// TwinCAT 3 PLC project rixs_optics_sim
// ProgramVersion: 3.1.4022.7
// libraries:
//   lcls2-cc-lib, * (SLAC)
//   PMPS, * (SLAC - LCLS)
//   Tc2_MC2, * (Beckhoff Automation GmbH)
//   Tc2_SerialCom, * (Beckhoff Automation GmbH)
//   Tc2_Standard, * (Beckhoff Automation GmbH)
//   Tc2_System, * (Beckhoff Automation GmbH)
//   Tc2_TcpIp, * (Beckhoff Automation GmbH)
//   Tc2_Utilities, * (Beckhoff Automation GmbH)
//   Tc3_Module, * (Beckhoff Automation GmbH)
//   LCLS General,newest,SLAC
//   lcls-twincat-motion,newest,SLAC
//   lcls-twincat-optics,newest,SLAC
// project tree:
//   DUTs/ ENUM_XS_YAG_States.TcDUT (not stored)
//   Function Blocks/ FB_XS_YAG_States.TcPOU (not stored)
//   GVLs/ GVL_COM_Buffers.TcGVL (not stored), GVL_M1K1.TcGVL (not stored), GVL_M1K1_BENDER_Constants.TcGVL (not stored), GVL_M1K1_BENDER_RTD.TcGVL (not stored), GVL_M1K1_Constants.TcGVL (not stored), GVL_M1K2.TcGVL (not stored), GVL_M1K2_Constants.TcGVL (not stored), GVL_PMPS.TcGVL, GVL_SerialIO.TcGVL (not stored), Main.TcGVL
//   / PiezoDriver.TcTTO (not stored), PlcTask.TcTTO (not stored), SerialIO.TcTTO (not stored)
//   POUs/DAQ Comm/ DUT_01_Channel_NW.TcDUT (not stored), DUT_Channel_NW.TcDUT (not stored), DUT_Header_NW.TcDUT (not stored), FB_AssembleChannel.TcPOU (not stored), FB_AssembleHeader.TcPOU (not stored), FB_UDPSocketHandler.TcPOU (not stored), F_AddChannelToHeader.TcPOU (not stored)
//   POUs/ PRG_1_PlcTask.TcPOU, PRG_2_PMPS_POST.TcPOU (not stored), PRG_DAQ_ENCODER.TcPOU (not stored), PRG_MR1K1_BEND.TcPOU, PRG_MR1K1_BEND_BENDER.TcPOU, PRG_MR1K2_SWITCH.TcPOU, PRG_SL1K2_EXIT.TcPOU, PRG_SP1K1_MONO.TcPOU, PRG_SPO_PMPS.TcPOU (not stored), PRG_ST1K1_ZOS.TcPOU (not stored), PRG_ZeroOrder_PMPS.TcPOU
//   POUs/Serial Comm/ PiezoSerial.TcPOU (not stored), P_Serial_Com.TcPOU (not stored)
//   Zero Order Functions/ F_Zbm1.TcPOU, F_Zbm3.TcPOU, F_hbm3.TcPOU, F_Theta_m3.TcPOU
// real-time tasks:
//   TASK PlcTask: cycle T#5ms, priority 20, ADS port 350
//   TASK PiezoDriver: cycle T#1ms, priority 3, ADS port 351
//   TASK SerialIO: cycle T#2ms, priority 1, ADS port 352
// motion (NC):
// I/O:
//   DEVICE Device 1 (EtherCAT)
// variable links:
//   rixs_optics_sim Instance <-> Device 1 (EtherCAT)/Term 1 (EK1200)/E5 (EK1122)/Box 84 (EP2338-0002)
//     PlcTask Outputs/PRG_SP1K1_MONO.bLEDPower01 <-> Channel 10/Output
//     PlcTask Outputs/PRG_SP1K1_MONO.bLEDPower02 <-> Channel 12/Output
//     PlcTask Outputs/PRG_SP1K1_MONO.bLEDPower03 <-> Channel 14/Output
//   rixs_optics_sim Instance <-> Device 1 (EtherCAT)/Term 1 (EK1200)/E5 (EK1122)/SL1K2-EXIT (EK1100)/EL5042_SL1K2_PITCH_VERT
//     PlcTask Inputs/Main.M19.nRawEncoderULINT <-> FB Inputs Channel 1/Position
//     PlcTask Inputs/Main.M20.nRawEncoderULINT <-> FB Inputs Channel 2/Position
//   rixs_optics_sim Instance <-> Device 1 (EtherCAT)/Term 1 (EK1200)/E5 (EK1122)/SL1K2-EXIT (EK1100)/EL5042_SL1K2_ROLL_GAP
//     PlcTask Inputs/Main.M21.nRawEncoderULINT <-> FB Inputs Channel 1/Position
//     PlcTask Inputs/Main.M22.nRawEncoderULINT <-> FB Inputs Channel 2/Position
//   rixs_optics_sim Instance <-> Device 1 (EtherCAT)/Term 1 (EK1200)/E5 (EK1122)/SL1K2-EXIT (EK1100)/EL5042_SL1K2_YAG
//     PlcTask Inputs/Main.M23.nRawEncoderULINT <-> FB Inputs Channel 1/Position
//   rixs_optics_sim Instance <-> Device 1 (EtherCAT)/Term 1 (EK1200)/E5 (EK1122)/SL1K2-EXIT (EK1100)/EL7047_SL1K2_GAP
//     PlcTask Inputs/Main.M22.bLimitBackwardEnable <-> STM Status/Status/Digital input 1
//     PlcTask Inputs/Main.M22.bLimitForwardEnable <-> STM Status/Status/Digital input 2
//   rixs_optics_sim Instance <-> Device 1 (EtherCAT)/Term 1 (EK1200)/E5 (EK1122)/SL1K2-EXIT (EK1100)/EL7047_SL1K2_PITCH
//     PlcTask Inputs/Main.M19.bLimitBackwardEnable <-> STM Status/Status/Digital input 1
//     PlcTask Inputs/Main.M19.bLimitForwardEnable <-> STM Status/Status/Digital input 2
//   rixs_optics_sim Instance <-> Device 1 (EtherCAT)/Term 1 (EK1200)/E5 (EK1122)/SL1K2-EXIT (EK1100)/EL7047_SL1K2_ROLL
//     PlcTask Inputs/Main.M21.bLimitBackwardEnable <-> STM Status/Status/Digital input 1
//     PlcTask Inputs/Main.M21.bLimitForwardEnable <-> STM Status/Status/Digital input 2
//   rixs_optics_sim Instance <-> Device 1 (EtherCAT)/Term 1 (EK1200)/E5 (EK1122)/SL1K2-EXIT (EK1100)/EL7047_SL1K2_VERT
//     PlcTask Inputs/Main.M20.bLimitBackwardEnable <-> STM Status/Status/Digital input 2
//     PlcTask Inputs/Main.M20.bLimitForwardEnable <-> STM Status/Status/Digital input 1
//   rixs_optics_sim Instance <-> Device 1 (EtherCAT)/Term 1 (EK1200)/E5 (EK1122)/SL1K2-EXIT (EK1100)/EL7047_SL1K2_YAG
//     PlcTask Inputs/Main.M23.bLimitBackwardEnable <-> STM Status/Status/Digital input 2
//     PlcTask Inputs/Main.M23.bLimitForwardEnable <-> STM Status/Status/Digital input 1
//   rixs_optics_sim Instance <-> Device 1 (EtherCAT)/Term 1 (EK1200)/E5 (EK1122)/X1 SP1K1-MONO(EK1100)/SP1K1-EL1004-E17
//     PlcTask Inputs/PRG_SP1K1_MONO.bSTOEnable1 <-> Channel 1/Input
//     PlcTask Inputs/PRG_SP1K1_MONO.bSTOEnable2 <-> Channel 2/Input
//   rixs_optics_sim Instance <-> Device 1 (EtherCAT)/Term 1 (EK1200)/E5 (EK1122)/X1 SP1K1-MONO(EK1100)/SP1K1-EL3054-E12
//     PlcTask Inputs/PRG_SP1K1_MONO.flow_1 <-> AI Standard Channel 1/Value
//     PlcTask Inputs/PRG_SP1K1_MONO.flow_2 <-> AI Standard Channel 2/Value
//     PlcTask Inputs/PRG_SP1K1_MONO.pres_1 <-> AI Standard Channel 3/Value
//   rixs_optics_sim Instance <-> Device 1 (EtherCAT)/Term 1 (EK1200)/E5 (EK1122)/X1 SP1K1-MONO(EK1100)/SP1K1-EL3202-E13
//     PlcTask Inputs/PRG_SP1K1_MONO.RTD1.bError <-> RTD Inputs Channel 1/Status/Error
//     PlcTask Inputs/PRG_SP1K1_MONO.RTD2.bError <-> RTD Inputs Channel 2/Status/Error
//     PlcTask Inputs/PRG_SP1K1_MONO.RTD1.bOverrange <-> RTD Inputs Channel 1/Status/Overrange
//     PlcTask Inputs/PRG_SP1K1_MONO.RTD2.bOverrange <-> RTD Inputs Channel 2/Status/Overrange
//     PlcTask Inputs/PRG_SP1K1_MONO.RTD1.bUnderrange <-> RTD Inputs Channel 1/Status/Underrange
//     PlcTask Inputs/PRG_SP1K1_MONO.RTD2.bUnderrange <-> RTD Inputs Channel 2/Status/Underrange
//     PlcTask Inputs/PRG_SP1K1_MONO.RTD1.iRaw <-> RTD Inputs Channel 1/Value
//     PlcTask Inputs/PRG_SP1K1_MONO.RTD2.iRaw <-> RTD Inputs Channel 2/Value
//   rixs_optics_sim Instance <-> Device 1 (EtherCAT)/Term 1 (EK1200)/E5 (EK1122)/X1 SP1K1-MONO(EK1100)/SP1K1-EL3202-E14
//     PlcTask Inputs/PRG_SP1K1_MONO.RTD3.bError <-> RTD Inputs Channel 1/Status/Error
//     PlcTask Inputs/PRG_SP1K1_MONO.RTD4.bError <-> RTD Inputs Channel 2/Status/Error
//     PlcTask Inputs/PRG_SP1K1_MONO.RTD3.bOverrange <-> RTD Inputs Channel 1/Status/Overrange
//     PlcTask Inputs/PRG_SP1K1_MONO.RTD4.bOverrange <-> RTD Inputs Channel 2/Status/Overrange
//     PlcTask Inputs/PRG_SP1K1_MONO.RTD3.bUnderrange <-> RTD Inputs Channel 1/Status/Underrange
//     PlcTask Inputs/PRG_SP1K1_MONO.RTD4.bUnderrange <-> RTD Inputs Channel 2/Status/Underrange
//     PlcTask Inputs/PRG_SP1K1_MONO.RTD3.iRaw <-> RTD Inputs Channel 1/Value
//     PlcTask Inputs/PRG_SP1K1_MONO.RTD4.iRaw <-> RTD Inputs Channel 2/Value
//   rixs_optics_sim Instance <-> Device 1 (EtherCAT)/Term 1 (EK1200)/E5 (EK1122)/X1 SP1K1-MONO(EK1100)/SP1K1-EL3204-E15
//     PlcTask Inputs/PRG_SP1K1_MONO.RTD5.bError <-> RTD Inputs Channel 1/Status/Error
//     PlcTask Inputs/PRG_SP1K1_MONO.RTD6.bError <-> RTD Inputs Channel 2/Status/Error
//     PlcTask Inputs/PRG_SP1K1_MONO.RTD5.bOverrange <-> RTD Inputs Channel 1/Status/Overrange
//     PlcTask Inputs/PRG_SP1K1_MONO.RTD6.bOverrange <-> RTD Inputs Channel 2/Status/Overrange
//     PlcTask Inputs/PRG_SP1K1_MONO.RTD5.bUnderrange <-> RTD Inputs Channel 1/Status/Underrange
//     PlcTask Inputs/PRG_SP1K1_MONO.RTD6.bUnderrange <-> RTD Inputs Channel 2/Status/Underrange
//     PlcTask Inputs/PRG_SP1K1_MONO.RTD5.iRaw <-> RTD Inputs Channel 1/Value
//     PlcTask Inputs/PRG_SP1K1_MONO.RTD6.iRaw <-> RTD Inputs Channel 2/Value
//   rixs_optics_sim Instance <-> Device 1 (EtherCAT)/Term 1 (EK1200)/E5 (EK1122)/X1 SP1K1-MONO(EK1100)/SP1K1-EL3204-E16
//     PlcTask Inputs/PRG_SP1K1_MONO.RTD7.bError <-> RTD Inputs Channel 1/Status/Error
//     PlcTask Inputs/PRG_SP1K1_MONO.RTD8.bError <-> RTD Inputs Channel 2/Status/Error
//     PlcTask Inputs/PRG_SP1K1_MONO.RTD7.bOverrange <-> RTD Inputs Channel 1/Status/Overrange
//     PlcTask Inputs/PRG_SP1K1_MONO.RTD8.bOverrange <-> RTD Inputs Channel 2/Status/Overrange
//     PlcTask Inputs/PRG_SP1K1_MONO.RTD7.bUnderrange <-> RTD Inputs Channel 1/Status/Underrange
//     PlcTask Inputs/PRG_SP1K1_MONO.RTD8.bUnderrange <-> RTD Inputs Channel 2/Status/Underrange
//     PlcTask Inputs/PRG_SP1K1_MONO.RTD7.iRaw <-> RTD Inputs Channel 1/Value
//     PlcTask Inputs/PRG_SP1K1_MONO.RTD8.iRaw <-> RTD Inputs Channel 2/Value
//   rixs_optics_sim Instance <-> Device 1 (EtherCAT)/Term 1 (EK1200)/E5 (EK1122)/X1 SP1K1-MONO(EK1100)/g_h_m
//     PlcTask Inputs/Main.M9.bLimitBackwardEnable <-> STM Status/Status/Digital input 2
//     PlcTask Inputs/Main.M9.bLimitForwardEnable <-> STM Status/Status/Digital input 1
//   rixs_optics_sim Instance <-> Device 1 (EtherCAT)/Term 1 (EK1200)/E5 (EK1122)/X1 SP1K1-MONO(EK1100)/g_pi_m
//     PlcTask Inputs/Main.M7.bLimitBackwardEnable <-> STM Status/Status/Digital input 2
//     PlcTask Inputs/Main.M7.bLimitForwardEnable <-> STM Status/Status/Digital input 1
//   rixs_optics_sim Instance <-> Device 1 (EtherCAT)/Term 1 (EK1200)/E5 (EK1122)/X1 SP1K1-MONO(EK1100)/g_pi_up_dwn_e
//     PlcTask Inputs/Main.M7.nRawEncoderULINT <-> FB Inputs Channel 2/Position
//     PlcTask Inputs/PRG_SP1K1_MONO.gpi_upe/Count <-> FB Inputs Channel 1/Position
//   rixs_optics_sim Instance <-> Device 1 (EtherCAT)/Term 1 (EK1200)/E5 (EK1122)/X1 SP1K1-MONO(EK1100)/m_h_e-g_h_e
//     PlcTask Inputs/Main.M8.nRawEncoderULINT <-> FB Inputs Channel 1/Position
//     PlcTask Inputs/Main.M9.nRawEncoderULINT <-> FB Inputs Channel 2/Position
//   rixs_optics_sim Instance <-> Device 1 (EtherCAT)/Term 1 (EK1200)/E5 (EK1122)/X1 SP1K1-MONO(EK1100)/m_h_m
//     PlcTask Inputs/Main.M8.bLimitBackwardEnable <-> STM Status/Status/Digital input 2
//     PlcTask Inputs/Main.M8.bLimitForwardEnable <-> STM Status/Status/Digital input 1
//   rixs_optics_sim Instance <-> Device 1 (EtherCAT)/Term 1 (EK1200)/E5 (EK1122)/X1 SP1K1-MONO(EK1100)/m_pi_m
//     PlcTask Inputs/Main.M6.bLimitBackwardEnable <-> STM Status/Status/Digital input 2
//     PlcTask Inputs/Main.M6.bLimitForwardEnable <-> STM Status/Status/Digital input 1
//   rixs_optics_sim Instance <-> Device 1 (EtherCAT)/Term 1 (EK1200)/E5 (EK1122)/X1 SP1K1-MONO(EK1100)/m_pi_up_dwn_e
//     PlcTask Inputs/Main.M6.nRawEncoderULINT <-> FB Inputs Channel 2/Position
//     PlcTask Inputs/PRG_SP1K1_MONO.mpi_upe/Count <-> FB Inputs Channel 1/Position
//   rixs_optics_sim Instance <-> Device 1 (EtherCAT)/Term 1 (EK1200)/E5 (EK1122)/X1 SP1K1-MONO(EK1100)/s_io_m
//     PlcTask Inputs/Main.M10.bLimitBackwardEnable <-> STM Status/Status/Digital input 2
//     PlcTask Inputs/Main.M10.bLimitForwardEnable <-> STM Status/Status/Digital input 1
//     PlcTask Inputs/Main.sio_current <-> STM Synchron info data/Info data 1
//     PlcTask Inputs/Main.sio_load <-> STM Synchron info data/Info data 2
//   rixs_optics_sim Instance <-> Device 1 (EtherCAT)/Term 1 (EK1200)/PMPS_FFO
//     PlcTask Outputs/GVL_PMPS.fbFastFaultOutput1.q_xFastFaultOut <-> Channel 1/Output
//     PlcTask Outputs/GVL_PMPS.fbFastFaultOutput2.q_xFastFaultOut <-> Channel 2/Output
//   rixs_optics_sim Instance <-> Device 1 (EtherCAT)/Term 1 (EK1200)/PMPS_PRE
//     PlcTask Inputs/PRG_2_PMPS_POST.fbArbiterIO.i_stCurrentBP <-> IO Inputs/CurrentBP
//     PlcTask Inputs/PRG_2_PMPS_POST.fbArbiterIO.xTxPDO_state <-> SYNC Inputs/TxPDO state
//     PlcTask Inputs/PRG_2_PMPS_POST.fbArbiterIO.xTxPDO_toggle <-> SYNC Inputs/TxPDO toggle
//     PlcTask Outputs/PRG_2_PMPS_POST.fbArbiterIO.q_stRequestedBP <-> IO Outputs/RequestedBP
//     PlcTask Outputs/PRG_MR1K1_BEND.nMR1K1_Y_ENC_PMPS <-> IO Outputs/MR1K1_Y_ENC
//   rixs_optics_sim Instance <-> Device 1 (EtherCAT)/Term 1 (EK1200)/Term 5 (EK1122)/EK1100_M1K2/EL5042_M1K2_Pitch
//     PlcTask Inputs/GVL_M1K1.M1K1_Pitch.diEncCnt <-> FB Inputs Channel 1/Position
//     PlcTask Inputs/GVL_M1K2.M1K2_Pitch.diEncCnt <-> FB Inputs Channel 1/Position
//   rixs_optics_sim Instance <-> Device 1 (EtherCAT)/Term 1 (EK1200)/Term 5 (EK1122)/EK1100_M1K2/EL6001_M1K2_PitchFine
//     SerialIO Inputs/GVL_SerialIO.Serial_stComIn_M1K2/D[{0..21}] <-> COM Inputs/Data In {0..21}  (22 links)
//     SerialIO Inputs/GVL_SerialIO.Serial_stComIn_M1K2/Status <-> COM Inputs/Status
//     SerialIO Outputs/GVL_SerialIO.Serial_stComOut_M1K2/Ctrl <-> COM Outputs/Ctrl
//     SerialIO Outputs/GVL_SerialIO.Serial_stComOut_M1K2/D[{0..21}] <-> COM Outputs/Data Out {0..21}  (22 links)
//   rixs_optics_sim Instance <-> Device 1 (EtherCAT)/Term 1 (EK1200)/Term 5 (EK1122)/EK1100_M1K2/EL7047_M1K2_PitchCoarse
//     PlcTask Inputs/Main.M5.bLimitBackwardEnable <-> STM Status/Status/Digital input 2
//     PlcTask Inputs/Main.M5.bLimitForwardEnable <-> STM Status/Status/Digital input 1
//   rixs_optics_sim Instance <-> Device 1 (EtherCAT)/Term 1 (EK1200)/Term 5 (EK1122)/EK1100_M1K2/EL7047_M1K2_Xdwn
//     PlcTask Inputs/Main.M4.bLimitBackwardEnable <-> STM Status/Status/Digital input 2
//     PlcTask Inputs/Main.M4.bLimitForwardEnable <-> STM Status/Status/Digital input 1
//   rixs_optics_sim Instance <-> Device 1 (EtherCAT)/Term 1 (EK1200)/Term 5 (EK1122)/EK1100_M1K2/EL7047_M1K2_Xup
//     PlcTask Inputs/Main.M3.bLimitBackwardEnable <-> STM Status/Status/Digital input 2
//     PlcTask Inputs/Main.M3.bLimitForwardEnable <-> STM Status/Status/Digital input 1
//   rixs_optics_sim Instance <-> Device 1 (EtherCAT)/Term 1 (EK1200)/Term 5 (EK1122)/EK1100_M1K2/EL7047_M1K2_Yleft
//     PlcTask Inputs/Main.M1.bLimitBackwardEnable <-> STM Status/Status/Digital input 2
//     PlcTask Inputs/Main.M1.bLimitForwardEnable <-> STM Status/Status/Digital input 1
//   rixs_optics_sim Instance <-> Device 1 (EtherCAT)/Term 1 (EK1200)/Term 5 (EK1122)/EK1100_M1K2/EL7047_M1K2_Yright
//     PlcTask Inputs/Main.M2.bLimitBackwardEnable <-> STM Status/Status/Digital input 2
//     PlcTask Inputs/Main.M2.bLimitForwardEnable <-> STM Status/Status/Digital input 1
//   rixs_optics_sim Instance <-> Device 1 (EtherCAT)/Term 1 (EK1200)/Term 5 (EK1122)/EK1100_MR1K1/EL1004_M1K1_STO
//     PlcTask Inputs/PRG_MR1K1_BEND.M1K1.fbRunHOMS.bSTOEnable1 <-> Channel 1/Input
//     PlcTask Inputs/PRG_MR1K1_BEND.M1K1.fbRunHOMS.bSTOEnable2 <-> Channel 2/Input
//   rixs_optics_sim Instance <-> Device 1 (EtherCAT)/Term 1 (EK1200)/Term 5 (EK1122)/EK1100_MR1K1/EL5042_M1K1_Pitch
//     PlcTask Inputs/Main.M16.nRawEncoderULINT <-> FB Inputs Channel 1/Position
//   rixs_optics_sim Instance <-> Device 1 (EtherCAT)/Term 1 (EK1200)/Term 5 (EK1122)/EK1100_MR1K1/EL5042_M1K1_Xupdwn
//     PlcTask Inputs/PRG_MR1K1_BEND.M1K1.fbRunHOMS.stXdwnEnc/Count <-> FB Inputs Channel 2/Position
//     PlcTask Inputs/PRG_MR1K1_BEND.M1K1.fbRunHOMS.stXupEnc/Count <-> FB Inputs Channel 1/Position
//   rixs_optics_sim Instance <-> Device 1 (EtherCAT)/Term 1 (EK1200)/Term 5 (EK1122)/EK1100_MR1K1/EL5042_M1K1_Yupdwn
//     PlcTask Inputs/Main.M12.nRawEncoderULINT <-> FB Inputs Channel 1/Position
//     PlcTask Inputs/PRG_MR1K1_BEND.M1K1.fbRunHOMS.stYdwnEnc/Count <-> FB Inputs Channel 2/Position
//     PlcTask Inputs/PRG_MR1K1_BEND.M1K1.fbRunHOMS.stYupEnc/Count <-> FB Inputs Channel 1/Position
//     PlcTask Inputs/PRG_MR1K1_BEND.bMR1K1_Y_ENC_Ready <-> FB Inputs Channel 1/Status/Ready
//     PlcTask Inputs/PRG_MR1K1_BEND.bMR1K1_Y_ENC_TxPDO <-> FB Inputs Channel 1/Status/TxPDO State
//   rixs_optics_sim Instance <-> Device 1 (EtherCAT)/Term 1 (EK1200)/Term 5 (EK1122)/EK1100_MR1K1/EL7047_M1K1_PitchCoarse
//     PlcTask Inputs/Main.M16.bLimitBackwardEnable <-> STM Status/Status/Digital input 2
//     PlcTask Inputs/Main.M16.bLimitForwardEnable <-> STM Status/Status/Digital input 1
//   rixs_optics_sim Instance <-> Device 1 (EtherCAT)/Term 1 (EK1200)/Term 5 (EK1122)/EK1100_MR1K1/EL7047_M1K1_Xdwn
//     PlcTask Inputs/Main.M15.bLimitBackwardEnable <-> STM Status/Status/Digital input 2
//     PlcTask Inputs/Main.M15.bLimitForwardEnable <-> STM Status/Status/Digital input 1
//   rixs_optics_sim Instance <-> Device 1 (EtherCAT)/Term 1 (EK1200)/Term 5 (EK1122)/EK1100_MR1K1/EL7047_M1K1_Xup
//     PlcTask Inputs/Main.M14.bLimitBackwardEnable <-> STM Status/Status/Digital input 2
//     PlcTask Inputs/Main.M14.bLimitForwardEnable <-> STM Status/Status/Digital input 1
//   rixs_optics_sim Instance <-> Device 1 (EtherCAT)/Term 1 (EK1200)/Term 5 (EK1122)/EK1100_MR1K1/EL7047_M1K1_Ydwn
//     PlcTask Inputs/Main.M12.bLimitBackwardEnable <-> STM Status/Status/Digital input 2
//     PlcTask Inputs/Main.M13.bLimitBackwardEnable <-> STM Status/Status/Digital input 2
//     PlcTask Inputs/Main.M13.bLimitForwardEnable <-> STM Status/Status/Digital input 1
//   rixs_optics_sim Instance <-> Device 1 (EtherCAT)/Term 1 (EK1200)/Term 5 (EK1122)/EK1100_MR1K1/EL7047_M1K1_Yup
//     PlcTask Inputs/Main.M12.bLimitForwardEnable <-> STM Status/Status/Digital input 1
//   rixs_optics_sim Instance <-> Device 1 (EtherCAT)/Term 1 (EK1200)/Term 5 (EK1122)/EK1100_MR1K1_BEND/EL1004_M1K1_BENDER_STO
//     PlcTask Inputs/PRG_MR1K1_BEND_BENDER.M1K1BENDbSTOEnable1 <-> Channel 1/Input
//     PlcTask Inputs/PRG_MR1K1_BEND_BENDER.M1K1BENDbSTOEnable2 <-> Channel 2/Input
//   rixs_optics_sim Instance <-> Device 1 (EtherCAT)/Term 1 (EK1200)/Term 5 (EK1122)/EK1100_MR1K1_BEND/EL2024-0010_M1K1_BEND_LED1
//     PlcTask Outputs/PRG_MR1K1_BEND.bLEDPower01 <-> Channel 1/Output
//     PlcTask Outputs/PRG_MR1K1_BEND.bLEDPower02 <-> Channel 2/Output
//     PlcTask Outputs/PRG_MR1K1_BEND.bLEDPower03 <-> Channel 3/Output
//     PlcTask Outputs/PRG_MR1K1_BEND.bLEDPower04 <-> Channel 4/Output
//   rixs_optics_sim Instance <-> Device 1 (EtherCAT)/Term 1 (EK1200)/Term 5 (EK1122)/EK1100_MR1K1_BEND/EL3202-0010_M1K1DS2_M1K1DS3
//     PlcTask Inputs/GVL_M1K1_BENDER_RTD.nM1K1DS_RTD_2 <-> RTD Inputs Channel 1/Value
//     PlcTask Inputs/GVL_M1K1_BENDER_RTD.nM1K1DS_RTD_3 <-> RTD Inputs Channel 2/Value
//   rixs_optics_sim Instance <-> Device 1 (EtherCAT)/Term 1 (EK1200)/Term 5 (EK1122)/EK1100_MR1K1_BEND/EL3202-0010_M1K1US1_M1K1US2
//     PlcTask Inputs/GVL_M1K1_BENDER_RTD.nM1K1US_RTD_1 <-> RTD Inputs Channel 1/Value
//     PlcTask Inputs/GVL_M1K1_BENDER_RTD.nM1K1US_RTD_2 <-> RTD Inputs Channel 2/Value
//   rixs_optics_sim Instance <-> Device 1 (EtherCAT)/Term 1 (EK1200)/Term 5 (EK1122)/EK1100_MR1K1_BEND/EL3202-0010_M1K1US3_M1K1DS1
//     PlcTask Inputs/GVL_M1K1_BENDER_RTD.nM1K1DS_RTD_1 <-> RTD Inputs Channel 2/Value
//     PlcTask Inputs/GVL_M1K1_BENDER_RTD.nM1K1US_RTD_3 <-> RTD Inputs Channel 1/Value
//   rixs_optics_sim Instance <-> Device 1 (EtherCAT)/Term 1 (EK1200)/Term 5 (EK1122)/EK1100_MR1K1_BEND/EL5042_M1K1_BEND_USDS
//     PlcTask Inputs/Main.M17.nRawEncoderULINT <-> FB Inputs Channel 1/Position
//     PlcTask Inputs/Main.M18.nRawEncoderULINT <-> FB Inputs Channel 2/Position
//   rixs_optics_sim Instance <-> Device 1 (EtherCAT)/Term 1 (EK1200)/Term 5 (EK1122)/EK1100_MR1K1_BEND/EL7041_M1K1_BEND_DS
//     PlcTask Inputs/Main.M18.bLimitBackwardEnable <-> STM Status/Status/Digital input 2
//     PlcTask Inputs/Main.M18.bLimitForwardEnable <-> STM Status/Status/Digital input 1
//   rixs_optics_sim Instance <-> Device 1 (EtherCAT)/Term 1 (EK1200)/Term 5 (EK1122)/EK1100_MR1K1_BEND/EL7041_M1K1_BEND_US
//     PlcTask Inputs/Main.M17.bLimitBackwardEnable <-> STM Status/Status/Digital input 2
//     PlcTask Inputs/Main.M17.bLimitForwardEnable <-> STM Status/Status/Digital input 1
//   rixs_optics_sim Instance <-> Device 1 (EtherCAT)/Term 1 (EK1200)/Term 5 (EK1122)/EK1100_ST1K2_ZOS/ST1K1-EL2008
//     PlcTask Outputs/Main.M24.bBrakeRelease <-> Channel 1/Output
//   rixs_optics_sim Instance <-> Device 1 (EtherCAT)/Term 1 (EK1200)/Term 5 (EK1122)/EK1100_ST1K2_ZOS/ST1K1-EL5042
//     PlcTask Inputs/Main.M24.nRawEncoderULINT <-> FB Inputs Channel 1/Position
//   rixs_optics_sim Instance <-> Device 1 (EtherCAT)/Term 1 (EK1200)/Term 5 (EK1122)/EK1100_ST1K2_ZOS/ST1K1-EL7041
//     PlcTask Inputs/Main.M24.bLimitBackwardEnable <-> STM Status/Status/Digital input 2
//     PlcTask Inputs/Main.M24.bLimitForwardEnable <-> STM Status/Status/Digital input 1
//   rixs_optics_sim Instance <-> NC-Task 1 SAF/Axes/Axis 24 ST1K1-ZOS-MMS
//     PlcTask Inputs/Main.M24.Axis.NcToPlc <-> Outputs/ToPlc
//     PlcTask Outputs/Main.M24.Axis.PlcToNc <-> Inputs/FromPlc
//   rixs_optics_sim Instance <-> NC-Task 1 SAF/Axes/M1K1-BEND-DS
//     PlcTask Inputs/Main.M18.Axis.NcToPlc <-> Outputs/ToPlc
//     PlcTask Outputs/Main.M18.Axis.PlcToNc <-> Inputs/FromPlc
//   rixs_optics_sim Instance <-> NC-Task 1 SAF/Axes/M1K1-BEND-US
//     PlcTask Inputs/Main.M17.Axis.NcToPlc <-> Outputs/ToPlc
//     PlcTask Outputs/Main.M17.Axis.PlcToNc <-> Inputs/FromPlc
//   rixs_optics_sim Instance <-> NC-Task 1 SAF/Axes/M1K1-Pitch
//     PlcTask Inputs/Main.M16.Axis.NcToPlc <-> Outputs/ToPlc
//     PlcTask Outputs/Main.M16.Axis.PlcToNc <-> Inputs/FromPlc
//   rixs_optics_sim Instance <-> NC-Task 1 SAF/Axes/M1K1-Xdwn
//     PlcTask Inputs/Main.M15.Axis.NcToPlc <-> Outputs/ToPlc
//     PlcTask Outputs/Main.M15.Axis.PlcToNc <-> Inputs/FromPlc
//   rixs_optics_sim Instance <-> NC-Task 1 SAF/Axes/M1K1-Xup
//     PlcTask Inputs/Main.M14.Axis.NcToPlc <-> Outputs/ToPlc
//     PlcTask Outputs/Main.M14.Axis.PlcToNc <-> Inputs/FromPlc
//   rixs_optics_sim Instance <-> NC-Task 1 SAF/Axes/M1K1-Ydwn
//     PlcTask Inputs/Main.M13.Axis.NcToPlc <-> Outputs/ToPlc
//     PlcTask Outputs/Main.M13.Axis.PlcToNc <-> Inputs/FromPlc
//   rixs_optics_sim Instance <-> NC-Task 1 SAF/Axes/M1K1-Yup
//     PlcTask Inputs/Main.M12.Axis.NcToPlc <-> Outputs/ToPlc
//     PlcTask Outputs/Main.M12.Axis.PlcToNc <-> Inputs/FromPlc
//   rixs_optics_sim Instance <-> NC-Task 1 SAF/Axes/M1K2-Pitch
//     PlcTask Inputs/Main.M5.Axis.NcToPlc <-> Outputs/ToPlc
//     PlcTask Outputs/Main.M5.Axis.PlcToNc <-> Inputs/FromPlc
//   rixs_optics_sim Instance <-> NC-Task 1 SAF/Axes/M1K2-Xdwn
//     PlcTask Inputs/Main.M4.Axis.NcToPlc <-> Outputs/ToPlc
//     PlcTask Outputs/Main.M4.Axis.PlcToNc <-> Inputs/FromPlc
//   rixs_optics_sim Instance <-> NC-Task 1 SAF/Axes/M1K2-Xup
//     PlcTask Inputs/Main.M3.Axis.NcToPlc <-> Outputs/ToPlc
//     PlcTask Outputs/Main.M3.Axis.PlcToNc <-> Inputs/FromPlc
//   rixs_optics_sim Instance <-> NC-Task 1 SAF/Axes/M1K2-Yleft
//     PlcTask Inputs/Main.M1.Axis.NcToPlc <-> Outputs/ToPlc
//     PlcTask Outputs/Main.M1.Axis.PlcToNc <-> Inputs/FromPlc
//   rixs_optics_sim Instance <-> NC-Task 1 SAF/Axes/M1K2-Yright
//     PlcTask Inputs/Main.M2.Axis.NcToPlc <-> Outputs/ToPlc
//     PlcTask Outputs/Main.M2.Axis.PlcToNc <-> Inputs/FromPlc
//   rixs_optics_sim Instance <-> NC-Task 1 SAF/Axes/SL1K2-CrystalGap-M22
//     PlcTask Inputs/Main.M22.Axis.NcToPlc <-> Outputs/ToPlc
//     PlcTask Outputs/Main.M22.Axis.PlcToNc <-> Inputs/FromPlc
//   rixs_optics_sim Instance <-> NC-Task 1 SAF/Axes/SL1K2-Pitch-M19
//     PlcTask Inputs/Main.M19.Axis.NcToPlc <-> Outputs/ToPlc
//     PlcTask Outputs/Main.M19.Axis.PlcToNc <-> Inputs/FromPlc
//   rixs_optics_sim Instance <-> NC-Task 1 SAF/Axes/SL1K2-Roll-M21
//     PlcTask Inputs/Main.M21.Axis.NcToPlc <-> Outputs/ToPlc
//     PlcTask Outputs/Main.M21.Axis.PlcToNc <-> Inputs/FromPlc
//   rixs_optics_sim Instance <-> NC-Task 1 SAF/Axes/SL1K2-Vert-M20
//     PlcTask Inputs/Main.M20.Axis.NcToPlc <-> Outputs/ToPlc
//     PlcTask Outputs/Main.M20.Axis.PlcToNc <-> Inputs/FromPlc
//   rixs_optics_sim Instance <-> NC-Task 1 SAF/Axes/SL1K2-YAG-M23
//     PlcTask Inputs/Main.M23.Axis.NcToPlc <-> Outputs/ToPlc
//     PlcTask Outputs/Main.M23.Axis.PlcToNc <-> Inputs/FromPlc
//   rixs_optics_sim Instance <-> NC-Task 1 SAF/Axes/g_h
//     PlcTask Inputs/Main.M9.Axis.NcToPlc <-> Outputs/ToPlc
//     PlcTask Outputs/Main.M9.Axis.PlcToNc <-> Inputs/FromPlc
//   rixs_optics_sim Instance <-> NC-Task 1 SAF/Axes/g_pi
//     PlcTask Inputs/Main.M7.Axis.NcToPlc <-> Outputs/ToPlc
//     PlcTask Outputs/Main.M7.Axis.PlcToNc <-> Inputs/FromPlc
//   rixs_optics_sim Instance <-> NC-Task 1 SAF/Axes/m_h
//     PlcTask Inputs/Main.M8.Axis.NcToPlc <-> Outputs/ToPlc
//     PlcTask Outputs/Main.M8.Axis.PlcToNc <-> Inputs/FromPlc
//   rixs_optics_sim Instance <-> NC-Task 1 SAF/Axes/m_pi
//     PlcTask Inputs/Main.M6.Axis.NcToPlc <-> Outputs/ToPlc
//     PlcTask Outputs/Main.M6.Axis.PlcToNc <-> Inputs/FromPlc
//   rixs_optics_sim Instance <-> NC-Task 1 SAF/Axes/s_io
//     PlcTask Inputs/Main.M10.Axis.NcToPlc <-> Outputs/ToPlc
//     PlcTask Outputs/Main.M10.Axis.PlcToNc <-> Inputs/FromPlc
//   rixs_optics_sim Instance <-> NC-Task 1 SAF/Axes/s_r
//     PlcTask Inputs/Main.M11.Axis.NcToPlc <-> Outputs/ToPlc
//     PlcTask Outputs/Main.M11.Axis.PlcToNc <-> Inputs/FromPlc

// ---- GVLs/GVL_PMPS.TcGVL
{attribute 'qualified_only'}
VAR_GLOBAL
	{attribute 'pytmc' := 'pv: SIM::RIX:OPTICS:ARB'}
    fbArbiter: FB_Arbiter(1);
    {attribute 'pytmc' := 'pv: SIM::RIX:OPTICS:FFO:01'}
    {attribute 'TcLinkTo' := '.q_xFastFaultOut:=TIIB[PMPS_FFO]^Channel 1^Output'}
    fbFastFaultOutput1: FB_HardwareFFOutput := (bAutoReset := TRUE);
    {attribute 'pytmc' := 'pv: SIM::RIX:OPTICS:FFO:02'}
    {attribute 'TcLinkTo' := '.q_xFastFaultOut:=TIIB[PMPS_FFO]^Channel 2^Output'}
    fbFastFaultOutput2: FB_HardwareFFOutput := (bAutoReset := TRUE);
	rPhotonEnergy :  REAL;
END_VAR

// ---- GVLs/Main.TcGVL
VAR_GLOBAL
(*
    Only includes motor definitions for the IOC
    These are hard-coded to be Main.M#,
    but are very convenient to store in a GVL,
    hence the confusing namespace here

    This should be refactored once the IOC
    supports arbitrary ads paths for motors
*)
	(*MR1K2*)
	// Motors
	{attribute 'TcLinkTo' := '.bLimitForwardEnable:=TIIB[EL7047_M1K2_Yleft]^STM Status^Status^Digital input 1;
                              .bLimitBackwardEnable:=TIIB[EL7047_M1K2_Yleft]^STM Status^Status^Digital input 2'}
	{attribute 'pytmc' := '
		pv: SIM:MR1K2:SWITCH:MMS:YLEFT
	'}
	M1 : DUT_MotionStage := (fVelocity:=100.0, nEnableMode:=ENUM_StageEnableMode.ALWAYS, bPowerSelf:=True); // M1K2 Yleft
	fbMotionStage_m1 : FB_MotionStage;

	{attribute 'TcLinkTo' := '.bLimitForwardEnable:=TIIB[EL7047_M1K2_Yright]^STM Status^Status^Digital input 1;
                              .bLimitBackwardEnable:=TIIB[EL7047_M1K2_Yright]^STM Status^Status^Digital input 2'}
	{attribute 'pytmc' := '
		pv: SIM:MR1K2:SWITCH:MMS:YRIGHT
	'}
	M2 : DUT_MotionStage := (fVelocity:=100.0, nEnableMode:=ENUM_StageEnableMode.ALWAYS, bPowerSelf:=True); // M1K2 Yright
	fbMotionStage_m2 : FB_MotionStage;

	{attribute 'TcLinkTo' := '.bLimitForwardEnable:=TIIB[EL7047_M1K2_Xup]^STM Status^Status^Digital input 1;
                              .bLimitBackwardEnable:=TIIB[EL7047_M1K2_Xup]^STM Status^Status^Digital input 2'}
	{attribute 'pytmc' := '
		pv: SIM:MR1K2:SWITCH:MMS:XUP
	'}
	M3 : DUT_MotionStage := (fVelocity:=150.0, nEnableMode:=ENUM_StageEnableMode.ALWAYS, bPowerSelf:=True); // M1K2 Xup
	fbMotionStage_m3 : FB_MotionStage;

	{attribute 'TcLinkTo' := '.bLimitForwardEnable:=TIIB[EL7047_M1K2_Xdwn]^STM Status^Status^Digital input 1;
                              .bLimitBackwardEnable:=TIIB[EL7047_M1K2_Xdwn]^STM Status^Status^Digital input 2'}
	{attribute 'pytmc' := '
		pv: SIM:MR1K2:SWITCH:MMS:XDWN
	'}
	M4 : DUT_MotionStage := (fVelocity:=150.0, nEnableMode:=ENUM_StageEnableMode.ALWAYS, bPowerSelf:=True); // M1K2 Xdwn
	fbMotionStage_m4 : FB_MotionStage;

	{attribute 'TcLinkTo' := '.bLimitForwardEnable:=TIIB[EL7047_M1K2_PitchCoarse]^STM Status^Status^Digital input 1;
                              .bLimitBackwardEnable:=TIIB[EL7047_M1K2_PitchCoarse]^STM Status^Status^Digital input 2'}
	{attribute 'pytmc' := '
		pv: SIM:MR1K2:SWITCH:MMS:PITCH
	'}
	M5 : DUT_MotionStage := (fVelocity:=30.0, nEnableMode:=ENUM_StageEnableMode.DURING_MOTION, bPowerSelf:=True); // M1K2 Pitch Stepper

	
	(*SP1K1-Mono*)
	{attribute 'pytmc' := '
		pv: SIM:SP1K1:MONO:MMS:M_PI
	'}
	{attribute 'TcLinkTo' := '.bLimitForwardEnable:=TIIB[m_pi_m]^STM Status^Status^Digital input 1;
                              .bLimitBackwardEnable:=TIIB[m_pi_m]^STM Status^Status^Digital input 2;
                              .nRawEncoderULINT:=TIIB[m_pi_up_dwn_e]^FB Inputs Channel 2^Position'}
	M6: DUT_MotionStage:=(nEnableMode:=ENUM_StageEnableMode.DURING_MOTION, fVelocity:=200.0, bPowerSelf:=True); // M_PI, urad
	{attribute 'pytmc' := '
		pv: SIM:SP1K1:MONO:MMS:G_PI
	'}
	{attribute 'TcLinkTo' := '.bLimitForwardEnable:=TIIB[g_pi_m]^STM Status^Status^Digital input 1;
                              .bLimitBackwardEnable:=TIIB[g_pi_m]^STM Status^Status^Digital input 2;
                              .nRawEncoderULINT:=TIIB[g_pi_up_dwn_e]^FB Inputs Channel 2^Position'}
	M7: DUT_MotionStage:=(nEnableMode:=ENUM_StageEnableMode.DURING_MOTION, fVelocity:=200.0, bPowerSelf:=True); // G_PI, urad
	{attribute 'pytmc' := '
		pv: SIM:SP1K1:MONO:MMS:M_H
	'}
	{attribute 'TcLinkTo' := '.bLimitForwardEnable:=TIIB[m_h_m]^STM Status^Status^Digital input 1;
                              .bLimitBackwardEnable:=TIIB[m_h_m]^STM Status^Status^Digital input 2;
							  .nRawEncoderULINT:=TIIB[m_h_e-g_h_e]^FB Inputs Channel 1^Position'}
	M8: DUT_MotionStage:=(nEnableMode:=ENUM_StageEnableMode.DURING_MOTION, fVelocity:=500.0, bPowerSelf:=True); // M_H, um
	{attribute 'pytmc' := '
		pv: SIM:SP1K1:MONO:MMS:G_H
	'}
	{attribute 'TcLinkTo' := '.bLimitForwardEnable:=TIIB[g_h_m]^STM Status^Status^Digital input 1;
                              .bLimitBackwardEnable:=TIIB[g_h_m]^STM Status^Status^Digital input 2;
							  .nRawEncoderULINT:=TIIB[m_h_e-g_h_e]^FB Inputs Channel 2^Position'}
	M9: DUT_MotionStage:=(nEnableMode:=ENUM_StageEnableMode.DURING_MOTION, fVelocity:=1000.0, bPowerSelf:=True); // G_H, um
	{attribute 'pytmc' := '
		pv: SIM:SP1K1:MONO:MMS:SD_V
	'}
	{attribute 'TcLinkTo' := '.bLimitForwardEnable:=TIIB[s_io_m]^STM Status^Status^Digital input 1;
                              .bLimitBackwardEnable:=TIIB[s_io_m]^STM Status^Status^Digital input 2'}
	M10: DUT_MotionStage:=(nEnableMode:=ENUM_StageEnableMode.DURING_MOTION, fVelocity:=500.0, bPowerSelf:=True); // SD_V, um
	{attribute 'pytmc' := '
		pv: SIM:SP1K1:MONO:MMS:SD_ROT
	'}
	// no limits on this motion
	M11: DUT_MotionStage:=(nEnableMode:=ENUM_StageEnableMode.DURING_MOTION, fVelocity:=500.0, bPowerSelf:=True); // SD_R, urad

	(*MR1K1*)
	// Should move before MR1K2 and re-number each motor, lots of work
    // need to fix Axis IDs for IOC to work
	// For now just want functional PLC project
	// Motors
	{attribute 'TcLinkTo' := '.bLimitForwardEnable:=TIIB[EL7047_M1K1_Yup]^STM Status^Status^Digital input 1;
                              .bLimitBackwardEnable:=TIIB[EL7047_M1K1_Ydwn]^STM Status^Status^Digital input 2;
							  .nRawEncoderULINT:=TIIB[EL5042_M1K1_Yupdwn]^FB Inputs Channel 1^Position'}
	{attribute 'pytmc' := '
		pv: SIM:MR1K1:BEND:MMS:YUP
	'}
	M12 : DUT_MotionStage := (fVelocity:=100.0, nEnableMode:=ENUM_StageEnableMode.ALWAYS, bPowerSelf:=True); // M1K1 Yup
	fbMotionStage_m12 : FB_MotionStage;

	{attribute 'TcLinkTo' := '.bLimitForwardEnable:=TIIB[EL7047_M1K1_Ydwn]^STM Status^Status^Digital input 1;
                              .bLimitBackwardEnable:=TIIB[EL7047_M1K1_Ydwn]^STM Status^Status^Digital input 2'}
	{attribute 'pytmc' := '
		pv: SIM:MR1K1:BEND:MMS:YDWN
	'}
	M13 : DUT_MotionStage := (fVelocity:=100.0, nEnableMode:=ENUM_StageEnableMode.ALWAYS, bPowerSelf:=True); // M1K1 Ydwn
	fbMotionStage_m13 : FB_MotionStage;

	{attribute 'TcLinkTo' := '.bLimitForwardEnable:=TIIB[EL7047_M1K1_Xup]^STM Status^Status^Digital input 1;
                              .bLimitBackwardEnable:=TIIB[EL7047_M1K1_Xup]^STM Status^Status^Digital input 2'}
	{attribute 'pytmc' := '
		pv: SIM:MR1K1:BEND:MMS:XUP
	'}
	M14 : DUT_MotionStage := (fVelocity:=150.0, nEnableMode:=ENUM_StageEnableMode.ALWAYS, bPowerSelf:=True); // M1K1 Xup
	fbMotionStage_m14 : FB_MotionStage;

	{attribute 'TcLinkTo' := '.bLimitForwardEnable:=TIIB[EL7047_M1K1_Xdwn]^STM Status^Status^Digital input 1;
                              .bLimitBackwardEnable:=TIIB[EL7047_M1K1_Xdwn]^STM Status^Status^Digital input 2'}
	{attribute 'pytmc' := '
		pv: SIM:MR1K1:BEND:MMS:XDWN
	'}
	M15 : DUT_MotionStage := (fVelocity:=150.0, nEnableMode:=ENUM_StageEnableMode.ALWAYS, bPowerSelf:=True); // M1K1 Xdwn
	fbMotionStage_m15 : FB_MotionStage;

	{attribute 'TcLinkTo' := '.bLimitForwardEnable:=TIIB[EL7047_M1K1_PitchCoarse]^STM Status^Status^Digital input 1;
                              .bLimitBackwardEnable:=TIIB[EL7047_M1K1_PitchCoarse]^STM Status^Status^Digital input 2;
                              .nRawEncoderULINT:=TIIB[EL5042_M1K1_Pitch]^FB Inputs Channel 1^Position'}
	{attribute 'pytmc' := '
		pv: SIM:MR1K1:BEND:MMS:PITCH
	'}
	M16 : DUT_MotionStage := (fVelocity:=30.0, nEnableMode:=ENUM_StageEnableMode.DURING_MOTION, bPowerSelf:=True); // M1K1 Pitch Stepper
		
	{attribute 'TcLinkTo' := '.bLimitForwardEnable :=TIIB[EL7041_M1K1_BEND_US]^STM Status^Status^Digital input 1;
                              .bLimitBackwardEnable:=TIIB[EL7041_M1K1_BEND_US]^STM Status^Status^Digital input 2;
							  .nRawEncoderULINT    := TIIB[EL5042_M1K1_BEND_USDS]^FB Inputs Channel 1^Position'}
	{attribute 'pytmc' := '
	pv: SIM:MR1K1:BEND:MMS:US
	'}
	M17 : DUT_MotionStage := (nEnableMode:=ENUM_StageEnableMode.DURING_MOTION, bPowerSelf:=TRUE); //MR1K1 US BEND
	fbMotionStage_m17 : FB_MotionStage;
	
	{attribute 'TcLinkTo' := '.bLimitForwardEnable :=TIIB[EL7041_M1K1_BEND_DS]^STM Status^Status^Digital input 1;
                              .bLimitBackwardEnable:=TIIB[EL7041_M1K1_BEND_DS]^STM Status^Status^Digital input 2;
							  .nRawEncoderULINT    := TIIB[EL5042_M1K1_BEND_USDS]^FB Inputs Channel 2^Position'}
	{attribute 'pytmc' := '
	pv: SIM:MR1K1:BEND:MMS:DS
	'}
	M18 : DUT_MotionStage := (nEnableMode:=ENUM_StageEnableMode.DURING_MOTION, bPowerSelf:=TRUE); //MR1K1 DS BEND
	fbMotionStage_m18 : FB_MotionStage;
	
	(*SL1K2*)
	// Motors
	{attribute 'TcLinkTo' := '.bLimitForwardEnable:=TIIB[EL7047_SL1K2_PITCH]^STM Status^Status^Digital input 2;
                              .bLimitBackwardEnable:=TIIB[EL7047_SL1K2_PITCH]^STM Status^Status^Digital input 1;
		 					  .nRawEncoderULINT      := TIIB[EL5042_SL1K2_PITCH_VERT]^FB Inputs Channel 1^Position'}
	{attribute 'pytmc' := '
		pv: SIM:SL1K2:EXIT:MMS:PITCH
	'}
	M19 : DUT_MotionStage := (sName:= 'SL1K2:EXIT:MMS:PITCH',fVelocity :=0.12);// Air Pitch

	{attribute 'TcLinkTo' := '.bLimitForwardEnable:=TIIB[EL7047_SL1K2_VERT]^STM Status^Status^Digital input 1;
                              .bLimitBackwardEnable:=TIIB[EL7047_SL1K2_VERT]^STM Status^Status^Digital input 2;
		 					  .nRawEncoderULINT      := TIIB[EL5042_SL1K2_PITCH_VERT]^FB Inputs Channel 2^Position'}
	{attribute 'pytmc' := '
		pv: SIM:SL1K2:EXIT:MMS:VERT
	'}
	M20 : DUT_MotionStage := (sName:= 'SL1K2:EXIT:MMS:VERT',fVelocity :=0.3); // Air Vertical

	{attribute 'TcLinkTo' := '.bLimitForwardEnable:=TIIB[EL7047_SL1K2_ROLL]^STM Status^Status^Digital input 2;
                              .bLimitBackwardEnable:=TIIB[EL7047_SL1K2_ROLL]^STM Status^Status^Digital input 1;
							  .nRawEncoderULINT      := TIIB[EL5042_SL1K2_ROLL_GAP]^FB Inputs Channel 1^Position'}
	{attribute 'pytmc' := '
		pv: SIM:SL1K2:EXIT:MMS:ROLL
	'}
	M21 : DUT_MotionStage := (sName:= 'SL1K2:EXIT:MMS:ROLL',fVelocity :=0.24); // Air Roll

	{attribute 'TcLinkTo' := '.bLimitForwardEnable:=TIIB[EL7047_SL1K2_GAP]^STM Status^Status^Digital input 2;
                              .bLimitBackwardEnable:=TIIB[EL7047_SL1K2_GAP]^STM Status^Status^Digital input 1;
							  .nRawEncoderULINT      := TIIB[EL5042_SL1K2_ROLL_GAP]^FB Inputs Channel 2^Position'}
	{attribute 'pytmc' := '
		pv: SIM:SL1K2:EXIT:MMS:GAP
	'}
	M22 : DUT_MotionStage := (sName:= 'SL1K2:EXIT:MMS:GAP',fVelocity :=0.1); // GAP

	{attribute 'TcLinkTo' := '.bLimitForwardEnable:=TIIB[EL7047_SL1K2_YAG]^STM Status^Status^Digital input 1;
                              .bLimitBackwardEnable:=TIIB[EL7047_SL1K2_YAG]^STM Status^Status^Digital input 2;
							  .nRawEncoderULINT      := TIIB[EL5042_SL1K2_YAG]^FB Inputs Channel 1^Position'}
	{attribute 'pytmc' := '
		pv: SIM:SL1K2:EXIT:MMS:YAG
	'}
	M23 : DUT_MotionStage := (sName:= 'SL1K2:EXIT:MMS:YAG',fVelocity :=0.5); // YAG
	
	
    // ST1K1-ZOS-MMS
    {attribute 'pytmc' := 'pv: SIM:ST1K1:ZOS:MMS'}
    {attribute 'TcLinkTo' := '.bLimitForwardEnable  := TIIB[ST1K1-EL7041]^STM Status^Status^Digital input 1;
                              .bLimitBackwardEnable := TIIB[ST1K1-EL7041]^STM Status^Status^Digital input 2;
							  .nRawEncoderULINT     :=TIIB[ST1K1-EL5042]^FB Inputs Channel 1^Position;
                              .bBrakeRelease        := TIIB[ST1K1-EL2008]^Channel 1^Output'}
    M24: DUT_MotionStage := (sName := 'ST1K1:ZOS:MMS');

	
	
	
	sio_current AT%I* : UINT;
	
	sio_load AT%I* : UINT;
	dummyBool: BOOL;
END_VAR

// ---- POUs/PRG_1_PlcTask.TcPOU
PROGRAM PRG_1_PlcTask
VAR

END_VAR

PRG_MR1K1_BEND();
PRG_MR1K1_BEND_BENDER();
//PRG_MR1K2_SWITCH();
PRG_SP1K1_MONO();
//PRG_SL1K2_EXIT();
PRG_ST1K1_ZOS();
//PRG_DAQ_ENCODER();
//PRG_SPO_PMPS();
PRG_2_PMPS_POST();

PRG_ZeroOrder_PMPS();

END_PROGRAM

// ---- POUs/PRG_MR1K1_BEND.TcPOU
PROGRAM PRG_MR1K1_BEND
VAR
	{attribute 'TcLinkTo' := '.fbRunHOMS.bSTOEnable1:=TIIB[EL1004_M1K1_STO]^Channel 1^Input;
                              .fbRunHOMS.bSTOEnable2:=TIIB[EL1004_M1K1_STO]^Channel 2^Input;
	                          .fbRunHOMS.stYupEnc.Count:=TIIB[EL5042_M1K1_Yupdwn]^FB Inputs Channel 1^Position;
	                          .fbRunHOMS.stYdwnEnc.Count:=TIIB[EL5042_M1K1_Yupdwn]^FB Inputs Channel 2^Position;
	                          .fbRunHOMS.stXupEnc.Count:=TIIB[EL5042_M1K1_Xupdwn]^FB Inputs Channel 1^Position;
	                          .fbRunHOMS.stXdwnEnc.Count:=TIIB[EL5042_M1K1_Xupdwn]^FB Inputs Channel 2^Position'}
	{attribute 'pytmc' := '
		pv: SIM:MR1K1:BEND
	'}
	M1K1 : DUT_HOMS;

	// Encoder Arrays/RMS Watch:
	{attribute 'pytmc' := '
		pv: SIM:MR1K1:BEND:ENC:Y
	'}
	fbYRMSErrorM1K1 : FB_RMSWatch;
	fMaxYRMSErrorM1K1 : LREAL;
	fMinYRMSErrorM1K1 : LREAL;

	{attribute 'pytmc' := '
		pv: SIM:MR1K1:BEND:ENC:X
	'}
	fbXRMSErrorM1K1 : FB_RMSWatch;
	fMaxXRMSErrorM1K1 : LREAL;
	fMinXRMSErrorM1K1 : LREAL;

	{attribute 'pytmc' := '
		pv: SIM:MR1K1:BEND:ENC:PITCH
	'}
	fbPitchRMSErrorM1K1 : FB_RMSWatch;
	fMaxPitchRMSErrorM1K1 : LREAL;
	fMinPitchRMSErrorM1K1 : LREAL;

	// Pitch Control
	fbM1K1PitchControl : FB_PitchControl;
	bM1K1PitchDone : BOOL;
	bM1K1PitchBusy : BOOL;

	// 3-15-20 Having issues with pitch control on new Axilon systems (M1K2)
	// Should test on this one to see if common to all new systems
	// Using stepper only for now
	fbMotionStage_m16 : FB_MotionStage;

	// Raw Encoder Counts
	{attribute 'pytmc' := '
		pv: SIM:MR1K1:BEND:ENC:YUP:CNT
		field: EGU cnt
		io: i
	'}
	nEncCntYupM1K1 : UDINT;
	{attribute 'pytmc' := '
		pv: SIM:MR1K1:BEND:ENC:YDWN:CNT
		field: EGU cnt
		io: i
	'}
	nEncCntYdwnM1K1 : UDINT;
	{attribute 'pytmc' := '
		pv: SIM:MR1K1:BEND:ENC:XUP:CNT
		field: EGU cnt
		io: i
	'}
	nEncCntXupM1K1 : UDINT;
	{attribute 'pytmc' := '
		pv: SIM:MR1K1:BEND:ENC:XDWN:CNT
		field: EGU cnt
		io: i
	'}
	nEncCntXdwnM1K1 : UDINT;
	{attribute 'pytmc' := '
		pv: SIM:MR1K1:BEND:ENC:PITCH:CNT
		field: EGU cnt
		io: i
	'}
	nEncCntPitchM1K1 : UDINT;

	// Encoder Reference Values
	{attribute 'pytmc' := '
		pv: SIM:MR1K1:BEND:ENC:YUP:REF
		field: EGU cnt
		io: i
	'}
	nEncRefYupM1K1 : UDINT;
	{attribute 'pytmc' := '
		pv: SIM:MR1K1:BEND:ENC:YDWN:REF
		field: EGU cnt
		io: i
	'}
	nEncRefYdwnM1K1 : UDINT;
	{attribute 'pytmc' := '
		pv: SIM:MR1K1:BEND:ENC:XUP:REF
		field: EGU cnt
		io: i
	'}
	nEncRefXupM1K1 : UDINT;
	{attribute 'pytmc' := '
		pv: SIM:MR1K1:BEND:ENC:XDWN:REF
		field: EGU cnt
		io: i
	'}
	nEncRefXdwnM1K1 : UDINT;
	{attribute 'pytmc' := '
		pv: SIM:MR1K1:BEND:ENC:PITCH:REF
		field: EGU cnt
		io: i
	'}
	nEncRefPitchM1K1 : UDINT;
	mcReadParameterPitchM1K1 : MC_ReadParameter;
	fEncRefPitchM1K1_urad : LREAL; // Current Pitch encoder offset in urad

	// Common
	fEncLeverArm_mm : LREAL := 410.0;
	
	// Mirror LEDs
	{attribute 'pytmc' := '
        pv: SIM:MR1K1:BEND:LED:01:PWR
        io: io
        field: ZNAM OFF
        field: ONAM ON
    '}
	{attribute 'TcLinkTo' := 'TIIB[EL2024-0010_M1K1_BEND_LED1]^Channel 1^Output'}
    bLEDPower01 AT %Q*: BOOL;
	
	{attribute 'pytmc' := '
        pv: SIM:MR1K1:BEND:LED:02:PWR
        io: io
        field: ZNAM OFF
        field: ONAM ON
    '}
	{attribute 'TcLinkTo' := 'TIIB[EL2024-0010_M1K1_BEND_LED1]^Channel 2^Output'}
    bLEDPower02 AT %Q*: BOOL;
			
	{attribute 'pytmc' := '
        pv: SIM:MR1K1:BEND:LED:03:PWR
        io: io
        field: ZNAM OFF
        field: ONAM ON
    '}
	{attribute 'TcLinkTo' := 'TIIB[EL2024-0010_M1K1_BEND_LED1]^Channel 3^Output'}
    bLEDPower03 AT %Q*: BOOL;
	{attribute 'pytmc' := '
        pv: SIM:MR1K1:BEND:LED:04:PWR
        io: io
        field: ZNAM OFF
        field: ONAM ON
    '}
	{attribute 'TcLinkTo' := 'TIIB[EL2024-0010_M1K1_BEND_LED1]^Channel 4^Output'}
    bLEDPower04 AT %Q*: BOOL;

    // MR1K1 Y Encoder for PMPS Veto Device
    ///////////////////////////////////////
        {attribute 'TcLinkTo' := 'TIIB[PMPS_PRE]^IO Outputs^MR1K1_Y_ENC'}
        nMR1K1_Y_ENC_PMPS AT %Q* : UDINT;
        {attribute 'TcLinkTo' := 'TIIB[EL5042_M1K1_Yupdwn]^FB Inputs Channel 1^Status^Ready'}
        bMR1K1_Y_ENC_Ready AT %I* : BOOL;
        {attribute 'TcLinkTo' := 'TIIB[EL5042_M1K1_Yupdwn]^FB Inputs Channel 1^Status^TxPDO State'}
        bMR1K1_Y_ENC_TxPDO AT %I* : BOOL;

END_VAR

// M1K1
M1K1.fbRunHOMS(stYup:=M12,
               stYdwn:=M13,
               stXup:=M14,
               stXdwn:=M15,
               stPitch:=M16,
	           nYupEncRef:=GVL_M1K1_Constants.nYUP_ENC_REF,
               nYdwnEncRef:=GVL_M1K1_Constants.nYDWN_ENC_REF,
               nXupEncRef:=GVL_M1K1_Constants.nXUP_ENC_REF,
               nXdwnEncRef:=GVL_M1K1_Constants.nXDWN_ENC_REF,
			   bExecuteCoupleY:=M1K1.bExecuteCoupleY,
               bExecuteCoupleX:=M1K1.bExecuteCoupleX,
			   bExecuteDecoupleY:=M1K1.bExecuteDecoupleY,
               bExecuteDecoupleX:=M1K1.bExecuteDecoupleX,
               bGantryAlreadyCoupledY=>M1K1.bGantryAlreadyCoupledY,
               bGantryAlreadyCoupledX=>M1K1.bGantryAlreadyCoupledX,
               nCurrGantryY=>M1K1.nCurrGantryY,
               nCurrGantryX=>M1K1.nCurrGantryX);

// No slave motion through Epics
M13.bExecute := FALSE; // M1K1-Ydwn
M15.bExecute := FALSE; // M1K1-Xdwn

// Convert nCurrGantry to um (smaller number) to read out in epics
M1K1.fCurrGantryY_um := LINT_TO_REAL(M1K1.nCurrGantryY) / 1000.0;
M1K1.fCurrGantryX_um := LINT_TO_REAL(M1K1.nCurrGantryX) / 1000.0;

// FB_MotionStage's for non-piezo axes
fbMotionStage_m12(stMotionStage:=M12);
fbMotionStage_m13(stMotionStage:=M13);
fbMotionStage_m14(stMotionStage:=M14);
fbMotionStage_m15(stMotionStage:=M15);

// Calculate Pitch RMS Error:
fbYRMSErrorM1K1(stMotionStage:=M12,
	            fMaxRMSError=>fMaxYRMSErrorM1K1,
				fMinRMSError=>fMinYRMSErrorM1K1);

fbXRMSErrorM1K1(stMotionStage:=M14,
	            fMaxRMSError=>fMaxXRMSErrorM1K1,
				fMinRMSError=>fMinXRMSErrorM1K1);

fbPitchRMSErrorM1K1(stMotionStage:=M16,
	                fMaxRMSError=>fMaxPitchRMSErrorM1K1,
					fMinRMSError=>fMinPitchRMSErrorM1K1);

(*
// Pitch Control
fbM1K1PitchControl(Pitch:=GVL_M1K1.M1K1_Pitch,
				   Stepper:=M16,
				   lrCurrentSetpoint:=M16.fPosition,
                   q_bDone=>bM1K1PitchDone,
                   q_bBusy=>bM1K1PitchBusy);
// When STO hit, need to reset SP
IF NOT M16.bHardwareEnable THEN
	M16.fPosition := M16.stAxisStatus.fActPosition;
END_IF
*)
// 3-15-20: Having issues with pitch control on new Axilon systems, should test here
fbMotionStage_m16(stMotionStage:=M16);

// Raw Encoder Counts For Epics
nEncCntYupM1K1 := ULINT_TO_UDINT(M1K1.fbRunHOMS.stYupEnc.Count);
nEncCntYdwnM1K1 := ULINT_TO_UDINT(M1K1.fbRunHOMS.stYdwnEnc.Count);
nEncCntXupM1K1 := ULINT_TO_UDINT(M1K1.fbRunHOMS.stXupEnc.Count);
nEncCntXdwnM1K1 := ULINT_TO_UDINT(M1K1.fbRunHOMS.stXdwnEnc.Count);
nEncCntPitchM1K1 := LINT_TO_UDINT(GVL_M1K1.M1K1_Pitch.diEncCnt);

// Encoder Reference Values For Epics
nEncRefYupM1K1 := ULINT_TO_UDINT(GVL_M1K1_Constants.nYUP_ENC_REF);
nEncRefYdwnM1K1 := ULINT_TO_UDINT(GVL_M1K1_Constants.nYDWN_ENC_REF);
nEncRefXupM1K1 := ULINT_TO_UDINT(GVL_M1K1_Constants.nXUP_ENC_REF);
nEncRefXdwnM1K1 := ULINT_TO_UDINT(GVL_M1K1_Constants.nXDWN_ENC_REF);
mcReadParameterPitchM1K1(Axis:=M16.Axis,
	                     Enable:=TRUE,
				         ParameterNumber:=MC_AxisParameter.AxisEncoderOffset,
				         ReadMode:=READMODE_CYCLIC,
				         Value=>fEncRefPitchM1K1_urad);

nEncRefPitchM1K1 := LREAL_TO_UDINT(ABS(fEncRefPitchM1K1_urad) * fEncLeverArm_mm);

// Export the Y encoder value for PMPS veto device evaluation
    IF bMR1K1_Y_ENC_Ready AND NOT bMR1K1_Y_ENC_TxPDO THEN
        nMR1K1_Y_ENC_PMPS := nEncCntYupM1K1;
    ELSE
        nMR1K1_Y_ENC_PMPS := 0;
    END_IF

END_PROGRAM

// ---- POUs/PRG_MR1K1_BEND_BENDER.TcPOU
PROGRAM PRG_MR1K1_BEND_BENDER
VAR
	// Encoder Arrays/RMS Watch:
	//MR1K1 US BENDER ENC RMS
	{attribute 'pytmc' := '
		pv: SIM:MR1K1:BEND:ENC:US
	'}
	fbBendUSRMSErrorM1K1 : FB_RMSWatch;
	fMaxBendUSRMSErrorM1K1 : LREAL;
	fMinBendUSRMSErrorM1K1 : LREAL;	
	//MR1K1 DS BENDER ENC RMS
	{attribute 'pytmc' := '
		pv: SIM:MR1K1:BEND:ENC:DS
	'}
	fbBendDSRMSErrorM1K1 : FB_RMSWatch;
	fMaxBendDSRMSErrorM1K1 : LREAL;
	fMinBendDSRMSErrorM1K1 : LREAL;

	// Encoder Reference Values
	//MR1K1 BEND US ENC REF
	{attribute 'pytmc' := '
		pv: SIM:MR1K1:BEND:ENC:US:REF
		field: EGU cnt
		io: i
	'}
	nEncRefBendUSM1K1 : UDINT;
	//MR1K1 BEND DS ENC REF
	{attribute 'pytmc' := '
		pv: SIM:MR1K1:BEND:ENC:DS:REF
		field: EGU cnt
		io: i
	'}
	nEncRefBendDSM1K1 : UDINT;
	
	// Encoder raw counts
	//M1K1 BEND US ENC CNT
	{attribute 'pytmc' := '
		pv: SIM:MR1K1:BEND:ENC:US:CNT
		field: EGU cnt
		io: i
	'}
	nEncCntBendUSM1K1 : UDINT;
	//M1K1 BEND DS ENC CNT
	{attribute 'pytmc' := '
		pv: SIM:MR1K1:BEND:ENC:DS:CNT
		field: EGU cnt
		io: i
	'}
	nEncCntBendDSM1K1 : UDINT;
	//Emergency Stop for MR1K1
	//Emergency Stop for MR1K1
	{attribute 'TcLinkTo' := 'TIID^Device 1 (EtherCAT)^Term 1 (EK1200)^Term 5 (EK1122)^EK1100_MR1K1_BEND^EL1004_M1K1_BENDER_STO^Channel 1^Input'}
	M1K1BENDbSTOEnable1 AT %I* : BOOL;
	{attribute 'TcLinkTo' := 'TIID^Device 1 (EtherCAT)^Term 1 (EK1200)^Term 5 (EK1122)^EK1100_MR1K1_BEND^EL1004_M1K1_BENDER_STO^Channel 2^Input'}
	M1K1BENDbSTOEnable2 AT %I* : BOOL;

	// MR1K1 Bender RTDs
	// MR1K1 US RTDs
	{attribute 'pytmc' := '
		pv: SIM:MR1K1:BEND:RTD:US:1
		field: ASLO 0.01
		field: EGU C
		io: i
	'}
	fM1K1US_RTD_1 : REAL;
	{attribute 'pytmc' := '
		pv: SIM:MR1K1:BEND:RTD:US:2
		field: ASLO 0.01
		field: EGU C
		io: i
	'}
	fM1K1US_RTD_2 : REAL;
	{attribute 'pytmc' := '
		pv: SIM:MR1K1:BEND:RTD:US:3
		field: ASLO 0.01
		field: EGU C
		io: i
	'}
	fM1K1US_RTD_3 : REAL;

	// M1K1 DS RTDs
	{attribute 'pytmc' := '
		pv: SIM:MR1K1:BEND:RTD:DS:1
		field: ASLO 0.01
		field: EGU C
		io: i
	'}
	fM1K1DS_RTD_1 : REAL;
	{attribute 'pytmc' := '
		pv: SIM:MR1K1:BEND:RTD:DS:2
		field: ASLO 0.01
		field: EGU C
		io: i
	'}
	fM1K1DS_RTD_2 : REAL;
	{attribute 'pytmc' := '
		pv: SIM:MR1K1:BEND:RTD:DS:3
		field: ASLO 0.01
		field: EGU C
		io: i
	'}
	fM1K1DS_RTD_3 : REAL;
	
	// RTD error bit
	bM1K1US_RTD_1_Err AT %I*: BOOL;
	bM1K1US_RTD_2_Err AT %I*: BOOL;
	bM1K1US_RTD_3_Err AT %I*: BOOL;
	bM1K1DS_RTD_1_Err AT %I*: BOOL;
	bM1K1DS_RTD_2_Err AT %I*: BOOL;
	bM1K1DS_RTD_3_Err AT %I*: BOOL;

	// Logging
	fbLogHandler : FB_LogHandler;
	fbBendUSRMSErrorMR1K1: INT;
    
    // PMPS
    ffBenderRange : FB_FastFault := (
        i_xAutoReset := TRUE,
        i_DevName := 'MR1K1 Bender',
        i_Desc := 'Benders have moved out of range, monochromator beam may be focused where it can damage the BCS. Adjust bender to be within limits to clear fault',
        i_TypeCode := 16#402);
END_VAR

//FB_Motion stages for MR1K1 Benders
//MR1K1 BEND
fbMotionStage_m17(stMotionStage:=M17);
fbMotionStage_m18(stMotionStage:=M18);

// Calculate Pitch RMS Error for MR1K1 Benders:
//MR1K1 US BENDER ENC RMS
fbBendUSRMSErrorM1K1(stMotionStage:=M17,
					 fMaxRMSError=>fMaxBendUSRMSErrorM1K1,
					 fMinRMSError=>fMinBendUSRMSErrorM1K1);
//MR1K1 DS BENDER ENC RMS
fbBendDSRMSErrorM1K1(stMotionStage:=M18,
					 fMaxRMSError=>fMaxBendDSRMSErrorM1K1,
					 fMinRMSError=>fMinBendDSRMSErrorM1K1);
					 
					 
//STO for MR1K1 Benders
M17.bHardwareEnable := M1K1BENDbSTOEnable1 AND M1K1BENDbSTOEnable2;
M18.bHardwareEnable := M1K1BENDbSTOEnable1 AND M1K1BENDbSTOEnable2;

//Encoder reference positions for MR1K1
nEncRefBendUSM1K1  := ULINT_TO_UDINT(GVL_M1K1_BENDER_Constants.nM1K1bendUS_ENC_REF);
nEncRefBendDSM1K1  := ULINT_TO_UDINT(GVL_M1K1_BENDER_Constants.nM1K1bendDS_ENC_REF);

// M1K1 Bender Encoder Count Values For Epics
nEncCntBendUSM1K1  := ULINT_TO_UDINT(M17.nRawEncoderULINT);
nEncCntBendDSM1K1  := ULINT_TO_UDINT(M18.nRawEncoderULINT);	

// MR1K1 Bender RTDs
fM1K1US_RTD_1 := INT_TO_REAL(GVL_M1K1_BENDER_RTD.nM1K1US_RTD_1);
fM1K1US_RTD_2 := INT_TO_REAL(GVL_M1K1_BENDER_RTD.nM1K1US_RTD_2);
fM1K1US_RTD_3 := INT_TO_REAL(GVL_M1K1_BENDER_RTD.nM1K1US_RTD_3);

fM1K1DS_RTD_1 := INT_TO_REAL(GVL_M1K1_BENDER_RTD.nM1K1DS_RTD_1);
fM1K1DS_RTD_2 := INT_TO_REAL(GVL_M1K1_BENDER_RTD.nM1K1DS_RTD_2);
fM1K1DS_RTD_3 := INT_TO_REAL(GVL_M1K1_BENDER_RTD.nM1K1DS_RTD_3);

// RTD not connected if T=0
(*
bM1K1US_RTD_1_Err := fM1K1US_RTD_1 = 0;
bM1K1US_RTD_2_Err := fM1K1DS_RTD_2 = 0;
bM1K1US_RTD_3_Err := fM1K1US_RTD_3 = 0;
bM1K1DS_RTD_1_Err := fM1K1DS_RTD_1 = 0;
bM1K1DS_RTD_2_Err := fM1K1DS_RTD_2 = 0;
bM1K1DS_RTD_3_Err := fM1K1DS_RTD_3 = 0;*)


// M1K1 Bender RTD interlocks
M17.bHardwareEnable R= fM1K1US_RTD_1 > 10000 OR bM1K1US_RTD_1_Err;
M18.bHardwareEnable R= fM1K1DS_RTD_1 > 10000 OR bM1K1DS_RTD_1_Err;

ffBenderRange.i_xOK :=
    GVL_M1K1_BENDER_Constants.nM1K1bendUS_PMPS_LowerLimit < nEncCntBendUSM1K1 AND nEncCntBendUSM1K1 < GVL_M1K1_BENDER_Constants.nM1K1bendUS_PMPS_UpperLimit AND
    GVL_M1K1_BENDER_Constants.nM1K1bendDS_PMPS_LowerLimit < nEncCntBendDSM1K1 AND nEncCntBendDSM1K1 < GVL_M1K1_BENDER_Constants.nM1K1bendDS_PMPS_UpperLimit;
ffBenderRange(io_fbFFHWO := GVL_PMPS.fbFastFaultOutput1);

END_PROGRAM

// ---- POUs/PRG_SP1K1_MONO.TcPOU
PROGRAM PRG_SP1K1_MONO
VAR
	
	// Where is the STO
	{attribute 'TcLinkTo' := 'TIID^Device 1 (EtherCAT)^Term 1 (EK1200)^E5 (EK1122)^X1 SP1K1-MONO(EK1100)^SP1K1-EL1004-E17^Channel 1^Input'}
	bSTOEnable1 AT %I*: BOOL;
	{attribute 'TcLinkTo' := 'TIID^Device 1 (EtherCAT)^Term 1 (EK1200)^E5 (EK1122)^X1 SP1K1-MONO(EK1100)^SP1K1-EL1004-E17^Channel 2^Input'}
	bSTOEnable2 AT %I*: BOOL;
	
	
	fbMotionStage_m_pi  :FB_MotionStage;
	fbMotionStage_g_pi  :FB_MotionStage;
	fbMotionStage_m_h   :FB_MotionStage;
	fbMotionStage_g_h   :FB_MotionStage;
	fbMotionStage_s_r   :FB_MotionStage;
	fbMotionStage_s_io  :FB_MotionStage;

	{attribute 'TcLinkTo' := '.Count:=TIIB[m_pi_up_dwn_e]^FB Inputs Channel 1^Position'}	
	mpi_upe  AT %I*:  ST_RenishawAbsEnc:=(ref:=0);
	{attribute 'TcLinkTo' := '.Count:=TIIB[g_pi_up_dwn_e]^FB Inputs Channel 1^Position'}
	gpi_upe  AT %I*:  ST_RenishawAbsEnc:=(ref:=0);

	{attribute 'pytmc' := '
		pv: SIM:SP1K1:MONO:ENC:M_PI:02
		io: o
	'}
	mpi_upeurad: LREAL;
	{attribute 'pytmc' := '
		pv: SIM:SP1K1:MONO:ENC:G_PI:02
		io: o
	'}
	gpi_upeurad: LREAL;
	
	
	(*Flow Switches*)
	{attribute 'TcLinkTo' := 'TIIB[SP1K1-EL3054-E12]^AI Standard Channel 1^Value'}
	flow_1 AT %I*: INT;
	{attribute 'TcLinkTo' := 'TIIB[SP1K1-EL3054-E12]^AI Standard Channel 2^Value'}	
	flow_2 AT %I*: INT;
	{attribute 'TcLinkTo' := 'TIIB[SP1K1-EL3054-E12]^AI Standard Channel 3^Value'}		
	pres_1 AT %I*: INT;
		
	{attribute 'pytmc' := '
		pv:  SIM:SP1K1:MONO:FSW:01
		io: o
	'}
	FLOW1 : LREAL := 0.00;
	
	{attribute 'pytmc' := '
		pv:  SIM:SP1K1:MONO:FSW:02
		io: o
	'}
	FLOW2 : LREAL := 0.00;
	
	{attribute 'pytmc' := '
		pv:  SIM:SP1K1:MONO:P1
		io: o
	'}
	PRES1 : LREAL := 0.00;


	(*RTDs*)
	{attribute 'pytmc' := '
		pv: SIM:SP1K1:MONO:RTD:01
		io: o
	'}
	 {attribute 'TcLinkTo' := '.iRaw := TIIB[SP1K1-EL3202-E13]^RTD Inputs Channel 1^Value;
                              .bError := TIIB[SP1K1-EL3202-E13]^RTD Inputs Channel 1^Status^Error;
                              .bUnderrange := TIIB[SP1K1-EL3202-E13]^RTD Inputs Channel 1^Status^Underrange;
                              .bOverrange := TIIB[SP1K1-EL3202-E13]^RTD Inputs Channel 1^Status^Overrange'}
	RTD1 : FB_TempSensor;
	
	{attribute 'pytmc' := '
		pv: SIM:SP1K1:MONO:RTD:02
		io: o
	'}
	{attribute 'TcLinkTo' := '.iRaw := TIIB[SP1K1-EL3202-E13]^RTD Inputs Channel 2^Value;
                              .bError := TIIB[SP1K1-EL3202-E13]^RTD Inputs Channel 2^Status^Error;
                              .bUnderrange := TIIB[SP1K1-EL3202-E13]^RTD Inputs Channel 2^Status^Underrange;
                              .bOverrange := TIIB[SP1K1-EL3202-E13]^RTD Inputs Channel 2^Status^Overrange'}
	RTD2 : FB_TempSensor;
	
	{attribute 'pytmc' := '
		pv: SIM:SP1K1:MONO:RTD:03
		io: o
	'}
	 {attribute 'TcLinkTo' := '.iRaw := TIIB[SP1K1-EL3202-E14]^RTD Inputs Channel 1^Value;
                              .bError := TIIB[SP1K1-EL3202-E14]^RTD Inputs Channel 1^Status^Error;
                              .bUnderrange := TIIB[SP1K1-EL3202-E14]^RTD Inputs Channel 1^Status^Underrange;
                              .bOverrange := TIIB[SP1K1-EL3202-E14]^RTD Inputs Channel 1^Status^Overrange'}
	RTD3 :FB_TempSensor;
	
	{attribute 'pytmc' := '
		pv: SIM:SP1K1:MONO:RTD:04
		io: o
	'}
	{attribute 'TcLinkTo' := '.iRaw := TIIB[SP1K1-EL3202-E14]^RTD Inputs Channel 2^Value;
                              .bError := TIIB[SP1K1-EL3202-E14]^RTD Inputs Channel 2^Status^Error;
                              .bUnderrange := TIIB[SP1K1-EL3202-E14]^RTD Inputs Channel 2^Status^Underrange;
                              .bOverrange := TIIB[SP1K1-EL3202-E14]^RTD Inputs Channel 2^Status^Overrange'}
	RTD4 : FB_TempSensor;
	
		{attribute 'pytmc' := '
		pv: SIM:SP1K1:MONO:RTD:05
		io: o
	'}
	{attribute 'TcLinkTo' := '.iRaw := TIIB[SP1K1-EL3204-E15]^RTD Inputs Channel 1^Value;
                              .bError := TIIB[SP1K1-EL3204-E15]^RTD Inputs Channel 1^Status^Error;
                              .bUnderrange := TIIB[SP1K1-EL3204-E15]^RTD Inputs Channel 1^Status^Underrange;
                              .bOverrange := TIIB[SP1K1-EL3204-E15]^RTD Inputs Channel 1^Status^Overrange'}
	RTD5 : FB_TempSensor;
	
	{attribute 'pytmc' := '
		pv: SIM:SP1K1:MONO:RTD:06
		io: o
	'}
	{attribute 'TcLinkTo' := '.iRaw := TIIB[SP1K1-EL3204-E15]^RTD Inputs Channel 2^Value;
                              .bError := TIIB[SP1K1-EL3204-E15]^RTD Inputs Channel 2^Status^Error;
                              .bUnderrange := TIIB[SP1K1-EL3204-E15]^RTD Inputs Channel 2^Status^Underrange;
                              .bOverrange := TIIB[SP1K1-EL3204-E15]^RTD Inputs Channel 2^Status^Overrange'}
	RTD6 : FB_TempSensor;
	
	{attribute 'pytmc' := '
		pv: SIM:SP1K1:MONO:RTD:07
		io: o
	'}
	{attribute 'TcLinkTo' := '.iRaw := TIIB[SP1K1-EL3204-E16]^RTD Inputs Channel 1^Value;
                              .bError := TIIB[SP1K1-EL3204-E16]^RTD Inputs Channel 1^Status^Error;
                              .bUnderrange := TIIB[SP1K1-EL3204-E16]^RTD Inputs Channel 1^Status^Underrange;
                              .bOverrange := TIIB[SP1K1-EL3204-E16]^RTD Inputs Channel 1^Status^Overrange'}
	RTD7 : FB_TempSensor;
	
	{attribute 'pytmc' := '
		pv: SIM:SP1K1:MONO:RTD:08
		io: o
	'}
	{attribute 'TcLinkTo' := '.iRaw := TIIB[SP1K1-EL3204-E16]^RTD Inputs Channel 2^Value;
                              .bError := TIIB[SP1K1-EL3204-E16]^RTD Inputs Channel 2^Status^Error;
                              .bUnderrange := TIIB[SP1K1-EL3204-E16]^RTD Inputs Channel 2^Status^Underrange;
                              .bOverrange := TIIB[SP1K1-EL3204-E16]^RTD Inputs Channel 2^Status^Overrange'}
	RTD8 :FB_TempSensor;
	
	
	
	
	
	//////////TODO
	
	{attribute 'pytmc' := '
		pv: SIM:GM:PITCH:fipi_read
		io: i
	'}	
	fipi_read: LREAL;
	
	{attribute 'pytmc' := '
		pv: SIM:GM:PITCH:fipi_set
		io: o
	'}
	fipi_set:  LREAL;
	
	{attribute 'pytmc' := '
        pv: SIM:SP1K1:MONO:LED:01:PWR
        io: io
        field: ZNAM OFF
        field: ONAM ON
    '}
	{attribute 'TcLinkTo' := 'TIID^Device 1 (EtherCAT)^Term 1 (EK1200)^E5 (EK1122)^Box 84 (EP2338-0002)^Channel 10^Output'}
    bLEDPower01 AT %Q*: BOOL;
	
	{attribute 'pytmc' := '
        pv: SIM:SP1K1:MONO:LED:02:PWR
        io: io
        field: ZNAM OFF
        field: ONAM ON
    '}
	{attribute 'TcLinkTo' := 'TIID^Device 1 (EtherCAT)^Term 1 (EK1200)^E5 (EK1122)^Box 84 (EP2338-0002)^Channel 12^Output'}
    bLEDPower02 AT %Q*: BOOL;
			
	{attribute 'pytmc' := '
        pv: SIM:SP1K1:MONO:LED:03:PWR
        io: io
        field: ZNAM OFF
        field: ONAM ON
    '}
	{attribute 'TcLinkTo' := 'TIID^Device 1 (EtherCAT)^Term 1 (EK1200)^E5 (EK1122)^Box 84 (EP2338-0002)^Channel 14^Output'}
    bLEDPower03 AT %Q*: BOOL;
	
	sd_io_FFO    :    FB_FastFault :=(
        i_DevName := 'SP1K1-MONO',
        i_Desc := 'Fault occurs When SP1K1-MONO screw driver motor is not in the out position',
        i_TypeCode := 16#1110);
	sd_io_e_pmps : LREAL:= 74000.29; 

END_VAR

// SP1K1-MONO
M6.bHardwareEnable := bSTOEnable1 AND bSTOEnable2;
M7.bHardwareEnable := bSTOEnable1 AND bSTOEnable2;
M8.bHardwareEnable := bSTOEnable1 AND bSTOEnable2; 
M9.bHardwareEnable := bSTOEnable1 AND bSTOEnable2;
M10.bHardwareEnable := bSTOEnable1 AND bSTOEnable2;
M11.bHardwareEnable := bSTOEnable1 AND bSTOEnable2;

fbMotionStage_m_pi  (stMotionStage:=M6);
fbMotionStage_g_pi  (stMotionStage:=M7);
fbMotionStage_m_h  (stMotionStage:=M8);
fbMotionStage_g_h  (stMotionStage:=M9);
fbMotionStage_s_io  (stMotionStage:=M10);
fbMotionStage_s_r  (stMotionStage:=M11);

//S_R with no hardware limit switched
M11.bLimitBackwardEnable := TRUE;
M11.bLimitForwardEnable := TRUE;

mpi_upeurad := ULINT_TO_LREAL(mpi_upe.Count)*0.004505;
gpi_upeurad := ULINT_TO_LREAL(gpi_upe.Count)*0.0066667;

(*Flow Switches and RTDs*)
FLOW1 := INT_TO_LREAL(flow_1)/32767*4;
FLOW2 := INT_TO_LREAL(flow_2)/32767*4;
PRES1 := INT_TO_LREAL(pres_1)/32767*2;
RTD1();
RTD2();
RTD3();
RTD4();
RTD5();
RTD6();
RTD7();
RTD8();

//Evaluate the encoder reading for the screw driver encoder. Fast fault when it is not out.
// i.e. encoder value must be greater than the out position (75000.29 - 1000u)
IF( M10.Axis.NcToPlc.ActPos < sd_io_e_pmps) THEN
        sd_io_FFO.i_xOK := FALSE;
    ELSE
        sd_io_FFO.i_xOK := TRUE;
END_IF

(*FAST FAULT*)
sd_io_FFO(i_xOK := ,
    i_xReset := ,
    i_xAutoReset :=TRUE,
    io_fbFFHWO := GVL_PMPS.fbFastFaultOutput1);

END_PROGRAM

// ---- POUs/PRG_ZeroOrder_PMPS.TcPOU
PROGRAM PRG_ZeroOrder_PMPS
VAR
	// PMPS
	ffZeroOrderBeam : FB_FastFault := (
        i_xAutoReset := TRUE,
        i_DevName := 'Zero Order Beam',
        i_Desc := 'Faults when Zero order beam safe conditions are not met',
        i_TypeCode := 16#F506);	
	{attribute 'pytmc' := '
        pv: SIM:SafeBenderRange
        field: ZNAM FALSE
        field: ONAM TRUE
    '}
    bSafeBenderRange : BOOL;
	
	{attribute 'pytmc' := '
        pv: SIM:LRG_Grating_IN
        field: ZNAM FALSE
        field: ONAM TRUE
    '}
    bLRG_Grating_IN : BOOL;
	
	{attribute 'pytmc' := '
        pv: SIM:ZOS_IN
        field: ZNAM FALSE
        field: ONAM TRUE
    '}
    bZOS_IN : BOOL;
	
	{attribute 'pytmc' := '
        pv: SIM:ZOB_on_Lower_Stopper
        field: ZNAM FALSE
        field: ONAM TRUE
    '}
    bZOB_on_Lower_Stopper : BOOL;
	
	{attribute 'pytmc' := '
        pv: SIM:MR1K1_Inserted
        field: ZNAM FALSE
        field: ONAM TRUE
    '}
    bMR1K1_Inserted : BOOL;
	
	{attribute 'pytmc' := '
        pv: SIM:ZeroOrderBeam
        field: ZNAM FALSE
        field: ONAM TRUE
    '}
    bZeroOrderBeam : BOOL;

END_VAR


ffZeroOrderBeam.i_xOK := SafeBenderRange() OR (LRG_Grating_IN() AND ZOS_IN() AND ZOB_on_Lower_Stopper() AND MR1K1_Inserted());
ffZeroOrderBeam(io_fbFFHWO := GVL_PMPS.fbFastFaultOutput1);


//Diagnostics
bSafeBenderRange := SafeBenderRange();
bLRG_Grating_IN := LRG_Grating_IN();
bZOS_IN := ZOS_IN();
bZOB_on_Lower_Stopper := ZOB_on_Lower_Stopper();
bMR1K1_Inserted := MR1K1_Inserted();
bZeroOrderBeam := ffZeroOrderBeam.i_xOK;

ACTION ACT_CALC:

END_ACTION

METHOD LRG_Grating_IN : BOOL
VAR_INPUT
END_VAR
LRG_Grating_IN := (M9.fPosition >= 24000) AND (M9.fPosition <= 28000);
END_METHOD

METHOD MR1K1_Inserted : BOOL
VAR_INPUT
END_VAR
MR1K1_Inserted := PMPS_GVL.stCurrentBeamParameters.aStoppers[PMPS.K_Stopper.MR1K1_IN] 
                    AND NOT PMPS_GVL.stCurrentBeamParameters.aStoppers[PMPS.K_Stopper.MR1K1_OUT];
END_METHOD

METHOD SafeBenderRange : BOOL
VAR_INPUT
END_VAR
 SafeBenderRange :=  GVL_M1K1_BENDER_Constants.nM1K1bendUS_PMPS_LowerLimit < M17.nEncoderCount AND M17.nEncoderCount < GVL_M1K1_BENDER_Constants.nM1K1bendUS_PMPS_UpperLimit AND
    GVL_M1K1_BENDER_Constants.nM1K1bendDS_PMPS_LowerLimit < M18.nEncoderCount AND M18.nEncoderCount < GVL_M1K1_BENDER_Constants.nM1K1bendDS_PMPS_UpperLimit;
END_METHOD

METHOD ZOB_on_Lower_Stopper : BOOL
VAR_INPUT
END_VAR
VAR
	Pm3 : LREAL;
	Pm2: LREAL;
	Pm1: LREAL;
	Hm1: LREAL;
	HZos:LREAL;
	Zbm1: LREAL;
	Zbm2: LREAL;
	Zbm3: LREAL;
	Hbm1: LREAL;
	Hbm2: LREAL;
	Hbm3: LREAL;
	Hb0m3:LREAL;
	//fixed calc
	Hm3	 : LREAL;
	Hpiv : LREAL;
	Theta_m1: LREAL;
	Theta_m2: LREAL;
	Theta_m3: LREAL;
	Delta : LREAL;
	Ans : LREAL;
END_VAR

VAR CONSTANT
	Hi2 :LREAL:=1.4;//m
	Zi2: LREAL :=731.613;//m
	Theta0 : LREAL:=0;
	Zm1 : LREAL:=733.772;//m
	Zmon : LREAL:=739.622;//m
	Zpiv : LREAL:= 739.622 ; //m
	Zzos : LREAL:= 741.422;//m
END_VAR


//Hm1 = 1400000+mr1k1 ben Y up
Hm1:= 1400000+M12.fPosition;
//Pm1 = 18310 - 281 + mr1k1 bend pitch 
Pm1 := 18310 - 281 + Main.M16.fPosition;
//Hpiv = 1.620305 + 0.001 // m 0.001 is correction from nominal
Hpiv:= 1.620305 + 0.001;
//Pm2 = mono mirror pitch - 90700 urad
Pm2 := Main.M6.fPosition - 90700;
//Hm3 = Hpiv + 0.006 m
Hm3:= Hpiv +0.006;
//Pm3 = mono grating pitch - 63300 urad
Pm3 := Main.M7.fPosition - 63300;
//Hzos = 1824.3 + st1k1_zos mm
Hzos:= 1824.3 + M24.fPosition;



Theta_m1 := 2*Pm1 - Theta0;
Theta_m2 := 2*Pm2 - Theta_m1;
Theta_m3 := 2 *Pm3 - 2 * Pm2 + 2* Pm1 - Theta0;


Zbm1 := (Hm1 - TAN(Pm1)* Zm1 - Hi2 + TAN(Theta0) *Zi2)/(TAN(Theta0) - TAN(Pm1));
hbm1 := TAN(Pm1)*Zbm1 + Hm1 - TAN(Pm1)*Zm1;

Zbm2 := (Hbm1 - TAN(Theta_m1)*Zbm1 - Hpiv + TAN(Pm2)*Zpiv)/ (TAN(Pm2) - TAN(Theta_m1));
Hbm2 := TAN(Pm2)*Zbm2 + Hpiv - TAN(Pm2)*Zpiv;

Zbm3 := (Hbm2 - TAN(Theta_m2)*Zbm2 - Hm3 + TAN(Pm3)*Zpiv)/ (TAN(Pm3) - TAN(Theta_m2));
Hbm3 := TAN(Pm3) * Zbm3 + Hm3 - TAN(Pm3)*Zpiv;

Hb0m3 := TAN(Theta_m3)*Zzos + Hbm3 - TAN(Theta_m3)*Zbm3;





//TRUE if hb0m3(Zzoz) - Hzos > D
Ans := Hb0m3 - Hzos;
IF GVL_PMPS.rPhotonEnergy <550 THEN
	ZOB_on_Lower_Stopper := Ans > 6;
	ELSIF GVL_PMPS.rPhotonEnergy <1000 THEN
		ZOB_on_Lower_Stopper := Ans >  3.2;
	ELSIF GVL_PMPS.rPhotonEnergy >=1000 THEN
		ZOB_on_Lower_Stopper := Ans >  2.5;	
		
END_IF
END_METHOD

METHOD ZOS_IN : BOOL
VAR_INPUT
END_VAR
IF GVL_PMPS.rPhotonEnergy >1500 THEN ZOS_IN:= FALSE;
	ELSIF (GVL_PMPS.rPhotonEnergy >1000 AND M24.fPosition>= 8.5) THEN ZOS_IN:= TRUE;
		ELSIF (GVL_PMPS.rPhotonEnergy <=1000 AND GVL_PMPS.rPhotonEnergy >550 AND M24.fPosition>= 7.9) THEN ZOS_IN:= TRUE;
			ELSIF (GVL_PMPS.rPhotonEnergy <=550 AND GVL_PMPS.rPhotonEnergy >200 AND M24.fPosition>= 6.9) THEN ZOS_IN:= TRUE;
				ELSE ZOS_IN:= FALSE;
END_IF
END_METHOD

END_PROGRAM

// ---- POUs/PRG_MR1K2_SWITCH.TcPOU
PROGRAM PRG_MR1K2_SWITCH
VAR
	{attribute 'TcLinkTo' := '.fbRunHOMS.bSTOEnable1:=TIIB[EL1004_M1K2_STO]^Channel 1^Input;
                              .fbRunHOMS.bSTOEnable2:=TIIB[EL1004_M1K2_STO]^Channel 2^Input;
	                          .fbRunHOMS.stYupEnc.Count:=TIIB[EL5042_M1K2_Yleftright]^FB Inputs Channel 1^Position;
	                          .fbRunHOMS.stYdwnEnc.Count:=TIIB[EL5042_M1K2_Yleftright]^FB Inputs Channel 2^Position;
	                          .fbRunHOMS.stXupEnc.Count:=TIIB[EL5042_M1K2_Xupdwn]^FB Inputs Channel 1^Position;
	                          .fbRunHOMS.stXdwnEnc.Count:=TIIB[EL5042_M1K2_Xupdwn]^FB Inputs Channel 2^Position'}
	{attribute 'pytmc' := '
		pv: SIM:MR1K2:SWITCH
	'}
	M1K2 : DUT_HOMS;

	// Encoder Arrays/RMS Watch:
	{attribute 'pytmc' := '
		pv: SIM:MR1K2:SWITCH:ENC:Y
	'}
	fbYRMSErrorM1K2 : FB_RMSWatch;
	fMaxYRMSErrorM1K2 : LREAL;
	fMinYRMSErrorM1K2 : LREAL;

	{attribute 'pytmc' := '
		pv: SIM:MR1K2:SWITCH:ENC:X
	'}
	fbXRMSErrorM1K2 : FB_RMSWatch;
	fMaxXRMSErrorM1K2 : LREAL;
	fMinXRMSErrorM1K2 : LREAL;

	{attribute 'pytmc' := '
		pv: SIM:MR1K2:SWITCH:ENC:PITCH
	'}
	fbPitchRMSErrorM1K2 : FB_RMSWatch;
	fMaxPitchRMSErrorM1K2 : LREAL;
	fMinPitchRMSErrorM1K2 : LREAL;

	// Pitch Control
	fbM1K2PitchControl : FB_PitchControl;
	bM1K2PitchDone : BOOL;
	bM1K2PitchBusy : BOOL;

	// 3-15-20 Having issues with pitch control on new Axilon systems
	// Using stepper only for now
	fbMotionStage_m5 : FB_MotionStage;
	
	// Roll (Rotation about Z axis) induced from Ygantry:
	{attribute 'pytmc' := '
		pv: SIM:MR1K2:SWITCH:ENC:ROLL
		field: EGU urad
		io: i
	'}
	fYRoll_urad : LREAL; // Roll about Z axis in urad

	// Raw Encoder Counts
	{attribute 'pytmc' := '
		pv: SIM:MR1K2:SWITCH:ENC:YLEFT:CNT
		field: EGU cnt
		io: i
	'}
	nEncCntYleftM1K2 : UDINT;
	{attribute 'pytmc' := '
		pv: SIM:MR1K2:SWITCH:ENC:YRIGHT:CNT
		field: EGU cnt
		io: i
	'}
	nEncCntYrightM1K2 : UDINT;
	{attribute 'pytmc' := '
		pv: SIM:MR1K2:SWITCH:ENC:XUP:CNT
		field: EGU cnt
		io: i
	'}
	nEncCntXupM1K2 : UDINT;
	{attribute 'pytmc' := '
		pv: SIM:MR1K2:SWITCH:ENC:XDWN:CNT
		field: EGU cnt
		io: i
	'}
	nEncCntXdwnM1K2 : UDINT;
	{attribute 'pytmc' := '
		pv: SIM:MR1K2:SWITCH:ENC:PITCH:CNT
		field: EGU cnt
		io: i
	'}
	nEncCntPitchM1K2 : UDINT;

	// Encoder Reference Values
	{attribute 'pytmc' := '
		pv: SIM:MR1K2:SWITCH:ENC:YLEFT:REF
		field: EGU cnt
		io: i
	'}
	nEncRefYleftM1K2 : UDINT;
	{attribute 'pytmc' := '
		pv: SIM:MR1K2:SWITCH:ENC:YRIGHT:REF
		field: EGU cnt
		io: i
	'}
	nEncRefYrightM1K2 : UDINT;
	{attribute 'pytmc' := '
		pv: SIM:MR1K2:SWITCH:ENC:XUP:REF
		field: EGU cnt
		io: i
	'}
	nEncRefXupM1K2 : UDINT;
	{attribute 'pytmc' := '
		pv: SIM:MR1K2:SWITCH:ENC:XDWN:REF
		field: EGU cnt
		io: i
	'}
	nEncRefXdwnM1K2 : UDINT;
	{attribute 'pytmc' := '
		pv: SIM:MR1K2:SWITCH:ENC:PITCH:REF
		field: EGU cnt
		io: i
	'}
	nEncRefPitchM1K2 : UDINT;
	mcReadParameterPitchM1K2 : MC_ReadParameter;
	fEncRefPitchM1K2_urad : LREAL; // Current Pitch encoder offset in urad

	// Common
	fEncLeverArm_mm : LREAL := 391.0;
END_VAR

// M1K2
M1K2.fbRunHOMS(stYup:=M1,
               stYdwn:=M2,
               stXup:=M3,
               stXdwn:=M4,
               stPitch:=M5,
	           nYupEncRef:=GVL_M1K2_Constants.nYLEFT_ENC_REF,
               nYdwnEncRef:=GVL_M1K2_Constants.nYRIGHT_ENC_REF,
               nXupEncRef:=GVL_M1K2_Constants.nXUP_ENC_REF,
               nXdwnEncRef:=GVL_M1K2_Constants.nXDWN_ENC_REF,
			   bExecuteCoupleY:=M1K2.bExecuteCoupleY,
               bExecuteCoupleX:=M1K2.bExecuteCoupleX,
			   bExecuteDecoupleY:=M1K2.bExecuteDecoupleY,
               bExecuteDecoupleX:=M1K2.bExecuteDecoupleX,
               bGantryAlreadyCoupledY=>M1K2.bGantryAlreadyCoupledY,
               bGantryAlreadyCoupledX=>M1K2.bGantryAlreadyCoupledX,
               nCurrGantryY=>M1K2.nCurrGantryY,
               nCurrGantryX=>M1K2.nCurrGantryX);

// No slave motion through Epics
M2.bExecute := FALSE; // M1K2-Yright
M4.bExecute := FALSE; // M1K2-Xdwn

// Convert nCurrGantry to um (smaller number) to read out in epics
M1K2.fCurrGantryY_um := LINT_TO_REAL(M1K2.nCurrGantryY) / 1000.0;
M1K2.fCurrGantryX_um := LINT_TO_REAL(M1K2.nCurrGantryX) / 1000.0;

fYRoll_urad := (REAL_TO_LREAL(ATAN(M1K2.fCurrGantryY_um / GVL_M1K2_Constants.fRollLeverArm_um))) * EXPT(10, 6);

// FB_MotionStage's for non-piezo axes
fbMotionStage_m1(stMotionStage:=M1);
fbMotionStage_m2(stMotionStage:=M2);
fbMotionStage_m3(stMotionStage:=M3);
fbMotionStage_m4(stMotionStage:=M4);

// Calculate Pitch RMS Error:
fbYRMSErrorM1K2(stMotionStage:=M1,
	            fMaxRMSError=>fMaxYRMSErrorM1K2,
				fMinRMSError=>fMinYRMSErrorM1K2);

fbXRMSErrorM1K2(stMotionStage:=M3,
	            fMaxRMSError=>fMaxXRMSErrorM1K2,
				fMinRMSError=>fMinXRMSErrorM1K2);

fbPitchRMSErrorM1K2(stMotionStage:=M5,
	                fMaxRMSError=>fMaxPitchRMSErrorM1K2,
					fMinRMSError=>fMinPitchRMSErrorM1K2);

(*
// Pitch Control
fbM1K2PitchControl(Pitch:=GVL_M1K2.M1K2_Pitch,
				   Stepper:=M5,
				   lrCurrentSetpoint:=M5.fPosition,
                   q_bDone=>bM1K2PitchDone,
                   q_bBusy=>bM1K2PitchBusy);
// When STO hit, need to reset SP
IF NOT M5.bHardwareEnable THEN
	M5.fPosition := M5.stAxisStatus.fActPosition;
END_IF
*)
// 3-15-20: Having issues with pitch control on new Axilon systems
fbMotionStage_m5(stMotionStage:=M5);

// Raw Encoder Counts For Epics
nEncCntYleftM1K2 := ULINT_TO_UDINT(M1K2.fbRunHOMS.stYupEnc.Count);
nEncCntYrightM1K2 := ULINT_TO_UDINT(M1K2.fbRunHOMS.stYdwnEnc.Count);
nEncCntXupM1K2 := ULINT_TO_UDINT(M1K2.fbRunHOMS.stXupEnc.Count);
nEncCntXdwnM1K2 := ULINT_TO_UDINT(M1K2.fbRunHOMS.stXdwnEnc.Count);
nEncCntPitchM1K2 := LINT_TO_UDINT(GVL_M1K2.M1K2_Pitch.diEncCnt);

// Encoder Reference Values For Epics
nEncRefYleftM1K2 := ULINT_TO_UDINT(GVL_M1K2_Constants.nYLEFT_ENC_REF);
nEncRefYrightM1K2 := ULINT_TO_UDINT(GVL_M1K2_Constants.nYRIGHT_ENC_REF);
nEncRefXupM1K2 := ULINT_TO_UDINT(GVL_M1K2_Constants.nXUP_ENC_REF);
nEncRefXdwnM1K2 := ULINT_TO_UDINT(GVL_M1K2_Constants.nXDWN_ENC_REF);
mcReadParameterPitchM1K2(Axis:=M5.Axis,
	                     Enable:=TRUE,
				         ParameterNumber:=MC_AxisParameter.AxisEncoderOffset,
				         ReadMode:=READMODE_CYCLIC,
				         Value=>fEncRefPitchM1K2_urad);

nEncRefPitchM1K2 := LREAL_TO_UDINT(ABS(fEncRefPitchM1K2_urad) * fEncLeverArm_mm);

END_PROGRAM

// ---- POUs/PRG_SL1K2_EXIT.TcPOU
PROGRAM PRG_SL1K2_EXIT
VAR
	FFO    :    FB_FastFault :=(
        i_DevName := 'SL1K2-EXIT',
        i_Desc := 'Fault occurs when device is in an usafe state',
        i_TypeCode := 16#E50);
	fbPitch: FB_MotionStage;
    fbRoll: FB_MotionStage;
    fbVertical: FB_MotionStage;
    fbGap: FB_MotionStage;
	fbYag: FB_MotionStage;
	
	 {attribute 'pytmc' := '
        pv: SIM:SL1K2:EXIT:YAG:STATE
        io: i
    '}
    fbStates: FB_XS_YAG_States;
	
	{attribute 'pytmc' := '
        pv: SIM:SL1K2:EXIT:RTD:CRYSTAL_TOP
    '}
    {attribute 'TcLinkTo' := '.iRaw := TIIB[EL3201_SL1K2_1]^RTD^Value;
                              .bError := TIIB[EL3201_SL1K2_1]^RTD^Status^Error;
                              .bUnderrange := TIIB[EL3201_SL1K2_1]^RTD^Status^Underrange;
                              .bOverrange := TIIB[EL3201_SL1K2_1]^RTD^Status^Overrange'}
    RTD_Crystal_TOP: FB_TempSensor;     
	{attribute 'pytmc' := '
        pv: SIM:SL1K2:EXIT:RTD:CRYSTAL_BOTTOM
    '}
    {attribute 'TcLinkTo' := '.iRaw := TIIB[EL3201_SL1K2_2]^RTD^Value;
                              .bError := TIIB[EL3201_SL1K2_2]^RTD^Status^Error;
                              .bUnderrange := TIIB[EL3201_SL1K2_2]^RTD^Status^Underrange;
                              .bOverrange := TIIB[EL3201_SL1K2_2]^RTD^Status^Overrange'}
    RTD_Crystal_BOTTOM: FB_TempSensor;   

	{attribute 'pytmc' := '
        pv: SIM:SL1K2:EXIT:RTD:YAG
    '}
    {attribute 'TcLinkTo' := '.iRaw := TIIB[EL3201_SL1K2_3]^RTD^Value;
                              .bError := TIIB[EL3201_SL1K2_3]^RTD^Status^Error;
                              .bUnderrange := TIIB[EL3201_SL1K2_3]^RTD^Status^Underrange;
                              .bOverrange := TIIB[EL3201_SL1K2_3]^RTD^Status^Overrange'}
    RTD_YAG: FB_TempSensor;    

	{attribute 'pytmc' := '
        pv: SIM:SL1K2:EXIT:RTD:HeatSync
    '}
    {attribute 'TcLinkTo' := '.iRaw := TIIB[EL3201_SL1K2_4]^RTD^Value;
                              .bError := TIIB[EL3201_SL1K2_4]^RTD^Status^Error;
                              .bUnderrange := TIIB[EL3201_SL1K2_4]^RTD^Status^Underrange;
                              .bOverrange := TIIB[EL3201_SL1K2_4]^RTD^Status^Overrange'}
    RTD_HeatSync: FB_TempSensor;      


	{attribute 'pytmc' := '
        pv: SIM:SL1K2:EXIT:FAN:PWR
		field: ZNAM OFF ;
		field: ONAM ON ;
    '}
	 {attribute 'TcLinkTo' := 'TIIB[EL2004_SL1K2]^Channel 1^Output'}
	bFanOn AT %Q*:BOOL;  

  {attribute 'pytmc' := '
        pv:  SIM:SL1K2:EXIT:LED:PWR
        io: io
        field: ZNAM OFF
        field: ONAM ON
    '}
	 {attribute 'TcLinkTo' := 'TIIB[EL2004_SL1K2]^Channel 2^Output'}
    bLEDPower AT %Q*: BOOL;   
	
	{attribute 'pytmc' := '
        pv: SIM:SL1K2:EXIT:CAM
    '}
	{attribute 'TcLinkTo' := '.iIlluminatorINT := TIIB[EL4004_SL1K2]^AO Outputs Channel 1^Analog output;
                              .bGigePower := TIIB[EL2004_SL1K2]^Channel 3^Output'}
    fbGige: FB_PPM_Gige;                 
	
	bInit : BOOL:=TRUE;
	
	 (*Motion Parameters*)
    fSmallDelta: LREAL := 0.01;
    fBigDelta: LREAL := 10;
    fMaxVelocity: LREAL := 0.5;
    fHighAccel: LREAL := 0.8;
    fLowAccel: LREAL := 0.1;
	
END_VAR

//  init the motion stages parameters
IF ( bInit) THEN
	bInit := FALSE;
	FFO.i_DevName := 'SL1K2-EXIT';
	//Pitch
    Main.M19.bHardwareEnable := TRUE;
    Main.M19.bPowerSelf :=TRUE;
    Main.M19.nBrakeMode := ENUM_StageBrakeMode.NO_BRAKE;
	Main.M19.nEnableMode := ENUM_StageEnableMode.DURING_MOTION;
   //Vert
	Main.M20.bHardwareEnable := TRUE;
    Main.M20.bPowerSelf :=TRUE;
    Main.M20.nBrakeMode := ENUM_StageBrakeMode.NO_BRAKE;
	Main.M20.nEnableMode := ENUM_StageEnableMode.DURING_MOTION;
	//ROLL
	Main.M21.bHardwareEnable := TRUE;
    Main.M21.bPowerSelf :=TRUE;
    Main.M21.nBrakeMode := ENUM_StageBrakeMode.NO_BRAKE;
	Main.M21.nEnableMode := ENUM_StageEnableMode.DURING_MOTION;
	//GAP
	Main.M22.bHardwareEnable := TRUE;
    Main.M22.bPowerSelf :=TRUE;
    Main.M22.nBrakeMode := ENUM_StageBrakeMode.NO_BRAKE;
	Main.M22.nEnableMode := ENUM_StageEnableMode.DURING_MOTION;
	//YAG
	Main.M23.bHardwareEnable := TRUE;
    Main.M23.bPowerSelf :=TRUE;
    Main.M23.nBrakeMode := ENUM_StageBrakeMode.NO_BRAKE;
	Main.M23.nEnableMode := ENUM_StageEnableMode.DURING_MOTION;
	
	// YAG STATES Parameters
	fbStates.nTransitionAssertionID := 16#E510;
	fbStates.nUnknownAssertionID := 16#E500;
	//Out
	fbStates.stOut.fPosition := 0;
	fbStates.stOut.bUseRawCounts := FALSE;
	fbStates.stOut.nRequestAssertionID := 16#E513;
	fbStates.stOut.stBeamParams := PMPS_GVL.cstFullBeam;
	fbStates.stOut.bValid := TRUE;
	//Yag1
	fbStates.stYag1.fPosition := 21;
	fbStates.stYag1.bUseRawCounts := FALSE;
	fbStates.stYag1.nRequestAssertionID := 16#E511;
	fbStates.stYag1.stBeamParams := PMPS_GVL.cstFullBeam;
	fbStates.stYag1.bValid := TRUE;
	//Yag2
	fbStates.stYag2.fPosition := 40;
	fbStates.stYag2.bUseRawCounts := FALSE;
	fbStates.stYag2.nRequestAssertionID := 16#E512;
	fbStates.stYag2.stBeamParams := PMPS_GVL.cstFullBeam;
	fbStates.stYag2.bValid := TRUE;
	
	//Turn on Fan by default
	bFanOn := TRUE;
END_IF



// Instantiate Function block for all the motion
fbPitch(stMotionStage:=Main.M19);//in Air
fbRoll(stMotionStage:=Main.M20);//in Air
fbVertical(stMotionStage:=Main.M21);//in Air
fbGap(stMotionStage:=Main.M22);//in vacuum
fbYag(stMotionStage:=Main.M23);//in vacuum


//States with PMPS
fbStates(
    fbArbiter:=GVL_PMPS.fbArbiter,
    fbFFHWO:=GVL_PMPS.fbFastFaultOutput1,
    nTransitionAssertionID:=,
    nUnknownAssertionID:=,
    stMotionStage:=Main.M23,
    bEnable:=TRUE,
    stOut:=,
    stYag1:=,
    stYag2:=);

//Camera and Ilumination
fbGige();
	
//RTDs
RTD_Crystal_TOP();
RTD_Crystal_BOTTOM();
RTD_YAG();
RTD_HeatSync();

END_PROGRAM

// ---- Zero Order Functions/F_Zbm1.TcPOU
FUNCTION F_Zbm1 : Real
VAR_INPUT
END_VAR
VAR
	Hm1: LREAL;
END_VAR
VAR CONSTANT
	bZm1 : REAL:=733.772//m
END_VAR

//Hm1 = 1400000+mr1k1 ben Y up
F_Hm1:= 1400000+M12.fPosition;

END_FUNCTION

// ---- Zero Order Functions/F_Zbm3.TcPOU
FUNCTION F_Zbm3 : REAL
VAR_INPUT
END_VAR
VAR
END_VAR

END_FUNCTION

// ---- Zero Order Functions/F_hbm3.TcPOU
FUNCTION F_hbm3 : REAL
VAR_INPUT
	Zbm: REAL;
END_VAR
VAR
	Pm3 : REAL;
	Hm3 : REAL;
END_VAR
VAR CONSTANT
	Zpiv : REAL:= 739.622 ; //m
	Hpiv : REAL:= 1.621305;//1.620305 + 0.001 // m 0.001 is correction from nominal
END_VAR


//Pm3 = mono grating pitch - 63300 urad
Pm3 := Main.M7.fPosition - 63300;

//hm3 = Hpiv + 0.006 m
Hm3 :=  Hpiv + 0.006;


F_hbm3 := TAN(Pm3) * Zbm + Hm3 - TAN(Pm3)*Zpiv;

END_FUNCTION

// ---- Zero Order Functions/F_Theta_m3.TcPOU
FUNCTION F_Theta_m3 : REAL
VAR_INPUT
END_VAR
VAR
	Pm3 : REAL;
	Pm2: REAL;
	Pm1: REAL;
	Theta0 : REAL:=0;
END_VAR



//Pm3 = mono grating pitch - 63300 urad
Pm3 := Main.M7.fPosition - 63300;

//Pm2 = mono mirror pitch - 90700 urad
Pm2 := Main.M6.fPosition - 90700;

//Pm1 = 18310 - 281 + mr1k1 bend pitch 
Pm1 := 18310 - 281 + Main.M16.fPosition;

F_Theta_m3 := 2 *Pm3 - 2 * Pm2 + 2* Pm1 - Theta0;

END_FUNCTION
